gfCNCPoint3[26390] = {X 477.0833, Y 62.5348, Z -4.6667, A 0.000, B 0.000, C 0.000 }
gfCNCPoint3[26391] = {X 476.2899, Y 62.8890, Z -4.6667, A 0.000, B 0.000, C 0.000 }
gfCNCPoint3[26392] = {X 475.4402, Y 63.0707, Z -4.6667, A 0.000, B 0.000, C 0.000 }
gfCNCPoint3[26393] = {X 475.4407, Y 92.8975, Z -4.6667, A 0.000, B 0.000, C 0.000 }
gfCNCPoint3[26394] = {X 475.8927, Y 93.0046, Z -4.6667, A 0.000, B 0.000, C 0.000 }
gfCNCPoint3[26395] = {X 476.3374, Y 93.1385, Z -4.6667, A 0.000, B 0.000, C 0.000 }
gfCNCPoint3[26396] = {X 477.1187, Y 93.4937, Z -4.6667, A 0.000, B 0.000, C 0.000 }
gfCNCPoint3[26397] = {X 477.8098, Y 94.0025, Z -4.6667, A 0.000, B 0.000, C 0.000 }
gfCNCPoint3[26398] = {X 478.3809, Y 94.6431, Z -4.6667, A 0.000, B 0.000, C 0.000 }
gfCNCPoint3[26399] = {X 478.8074, Y 95.3878, Z -4.6667, A 0.000, B 0.000, C 0.000 }
gfCNCPoint3[26400] = {X 479.0709, Y 96.2046, Z -4.6667, A 0.000, B 0.000, C 0.000 }
gfCNCPoint3[26401] = {X 479.1600, Y 97.0582, Z -4.6667, A 0.000, B 0.000, C 0.000 }
gfCNCPoint3[26402] = {X 479.1600, Y 98.0000, Z -4.6667, A 0.000, B 0.000, C 0.000 }
gfCNCPoint3[26403] = {X 479.0557, Y 98.9257, Z -4.6667, A 0.000, B 0.000, C 0.000 }
gfCNCPoint3[26404] = {X 478.7480, Y 99.8050, Z -4.6667, A 0.000, B 0.000, C 0.000 }
gfCNCPoint3[26405] = {X 478.2524, Y 100.5937, Z -4.6667, A 0.000, B 0.000, C 0.000 }
gfCNCPoint3[26406] = {X 477.5937, Y 101.2524, Z -4.6667, A 0.000, B 0.000, C 0.000 }
gfCNCPoint3[26407] = {X 476.8050, Y 101.7480, Z -4.6667, A 0.000, B 0.000, C 0.000 }
gfCNCPoint3[26408] = {X 475.9257, Y 102.0557, Z -4.6667, A 0.000, B 0.000, C 0.000 }
gfCNCPoint3[26409] = {X 475.0000, Y 102.1600, Z -4.6667, A 0.000, B 0.000, C 0.000 }
gfCNCPoint3[26410] = {X 458.4596, Y 102.1600, Z -4.6667, A 0.000, B 0.000, C 0.000 }
gfCNCPoint3[26411] = {X 457.5339, Y 102.0557, Z -4.6667, A 0.000, B 0.000, C 0.000 }
gfCNCPoint3[26412] = {X 456.6546, Y 101.7480, Z -4.6667, A 0.000, B 0.000, C 0.000 }
gfCNCPoint3[26413] = {X 455.8659, Y 101.2524, Z -4.6667, A 0.000, B 0.000, C 0.000 }
gfCNCPoint3[26414] = {X 455.2072, Y 100.5937, Z -4.6667, A 0.000, B 0.000, C 0.000 }
gfCNCPoint3[26415] = {X 454.7116, Y 99.8050, Z -4.6667, A 0.000, B 0.000, C 0.000 }
gfCNCPoint3[26416] = {X 454.4039, Y 98.9257, Z -4.6667, A 0.000, B 0.000, C 0.000 }
gfCNCPoint3[26417] = {X 454.2996, Y 98.0000, Z -4.6667, A 0.000, B 0.000, C 0.000 }
gfCNCPoint3[26418] = {X 454.2996, Y 97.0659, Z -4.6667, A 0.000, B 0.000, C 0.000 }
gfCNCPoint3[26419] = {X 454.3903, Y 96.2022, Z -4.6667, A 0.000, B 0.000, C 0.000 }
gfCNCPoint3[26420] = {X 454.6583, Y 95.3761, Z -4.6667, A 0.000, B 0.000, C 0.000 }
gfCNCPoint3[26421] = {X 455.0920, Y 94.6237, Z -4.6667, A 0.000, B 0.000, C 0.000 }
gfCNCPoint3[26422] = {X 455.6724, Y 93.9777, Z -4.6667, A 0.000, B 0.000, C 0.000 }
gfCNCPoint3[26423] = {X 456.3743, Y 93.4663, Z -4.6667, A 0.000, B 0.000, C 0.000 }
gfCNCPoint3[26424] = {X 457.1672, Y 93.1118, Z -4.6667, A 0.000, B 0.000, C 0.000 }
gfCNCPoint3[26425] = {X 458.0163, Y 92.9296, Z -4.6667, A 0.000, B 0.000, C 0.000 }
gfCNCPoint3[26426] = {X 458.0163, Y 85.4858, Z -4.6667, A 0.000, B 0.000, C 0.000 }
gfCNCPoint3[26427] = {X 444.8411, Y 80.3211, Z -4.6667, A 0.000, B 0.000, C 0.000 }
gfCNCPoint3[26428] = {X 419.8629, Y 96.5017, Z -4.6667, A 0.000, B 0.000, C 0.000 }
gfCNCPoint3[26429] = {X 419.8667, Y 97.0654, Z -4.6667, A 0.000, B 0.000, C 0.000 }
gfCNCPoint3[26430] = {X 419.8667, Y 98.0000, Z -4.6667, A 0.000, B 0.000, C 0.000 }
gfCNCPoint3[26431] = {X 419.7624, Y 98.9257, Z -4.6667, A 0.000, B 0.000, C 0.000 }
gfCNCPoint3[26432] = {X 419.4547, Y 99.8050, Z -4.6667, A 0.000, B 0.000, C 0.000 }
gfCNCPoint3[26433] = {X 418.9591, Y 100.5937, Z -4.6667, A 0.000, B 0.000, C 0.000 }
gfCNCPoint3[26434] = {X 418.3004, Y 101.2524, Z -4.6667, A 0.000, B 0.000, C 0.000 }
gfCNCPoint3[26435] = {X 417.5117, Y 101.7480, Z -4.6667, A 0.000, B 0.000, C 0.000 }
gfCNCPoint3[26436] = {X 416.6324, Y 102.0557, Z -4.6667, A 0.000, B 0.000, C 0.000 }
gfCNCPoint3[26437] = {X 415.7067, Y 102.1600, Z -4.6667, A 0.000, B 0.000, C 0.000 }
gfCNCPoint3[26438] = {X 396.4059, Y 102.1600, Z -4.6667, A 0.000, B 0.000, C 0.000 }
gfCNCPoint3[26439] = {X 395.4803, Y 102.0557, Z -4.6667, A 0.000, B 0.000, C 0.000 }
gfCNCPoint3[26440] = {X 394.6010, Y 101.7480, Z -4.6667, A 0.000, B 0.000, C 0.000 }
gfCNCPoint3[26441] = {X 393.8122, Y 101.2524, Z -4.6667, A 0.000, B 0.000, C 0.000 }
gfCNCPoint3[26442] = {X 393.1535, Y 100.5937, Z -4.6667, A 0.000, B 0.000, C 0.000 }
gfCNCPoint3[26443] = {X 392.6579, Y 99.8050, Z -4.6667, A 0.000, B 0.000, C 0.000 }
gfCNCPoint3[26444] = {X 392.3502, Y 98.9257, Z -4.6667, A 0.000, B 0.000, C 0.000 }
gfCNCPoint3[26445] = {X 392.2459, Y 98.0000, Z -4.6667, A 0.000, B 0.000, C 0.000 }
gfCNCPoint3[26446] = {X 392.2459, Y 97.0659, Z -4.6667, A 0.000, B 0.000, C 0.000 }
gfCNCPoint3[26447] = {X 392.3511, Y 96.1365, Z -4.6667, A 0.000, B 0.000, C 0.000 }
gfCNCPoint3[26448] = {X 392.6612, Y 95.2541, Z -4.6667, A 0.000, B 0.000, C 0.000 }
gfCNCPoint3[26449] = {X 393.1607, Y 94.4633, Z -4.6667, A 0.000, B 0.000, C 0.000 }
gfCNCPoint3[26450] = {X 393.8242, Y 93.8040, Z -4.6667, A 0.000, B 0.000, C 0.000 }
gfCNCPoint3[26451] = {X 394.6182, Y 93.3096, Z -4.6667, A 0.000, B 0.000, C 0.000 }
gfCNCPoint3[26452] = {X 395.5026, Y 93.0052, Z -4.6667, A 0.000, B 0.000, C 0.000 }
gfCNCPoint3[26453] = {X 396.4327, Y 92.9060, Z -4.6667, A 0.000, B 0.000, C 0.000 }
gfCNCPoint3[26454] = {X 397.3745, Y 92.8625, Z -4.6667, A 0.000, B 0.000, C 0.000 }
gfCNCPoint3[26455] = {X 398.3131, Y 92.7731, Z -4.6667, A 0.000, B 0.000, C 0.000 }
gfCNCPoint3[26456] = {X 398.9990, Y 92.6067, Z -4.6667, A 0.000, B 0.000, C 0.000 }
gfCNCPoint3[26457] = {X 399.6307, Y 92.2919, Z -4.6667, A 0.000, B 0.000, C 0.000 }
gfCNCPoint3[26458] = {X 413.8854, Y 83.1633, Z -4.6667, A 0.000, B 0.000, C 0.000 }
gfCNCPoint3[26459] = {X 411.7283, Y 79.7948, Z -4.6667, A 0.000, B 0.000, C 0.000 }
gfCNCPoint3[26460] = {X 413.9286, Y 83.2307, Z -4.6667, A 0.000, B 0.000, C 0.000 }
gfCNCPoint3[26461] = {X 428.5801, Y 73.8479, Z -4.6667, A 0.000, B 0.000, C 0.000 }
gfCNCPoint3[26462] = {X 403.8433, Y 64.1425, Z -4.6667, A 0.000, B 0.000, C 0.000 }
gfCNCPoint3[26463] = {X 402.1208, Y 63.5723, Z -4.6667, A 0.000, B 0.000, C 0.000 }
gfCNCPoint3[26464] = {X 400.3462, Y 63.1946, Z -4.6667, A 0.000, B 0.000, C 0.000 }
gfCNCPoint3[26465] = {X 398.5408, Y 63.0140, Z -4.6667, A 0.000, B 0.000, C 0.000 }
gfCNCPoint3[26466] = {X 397.6404, Y 62.9096, Z -4.6667, A 0.000, B 0.000, C 0.000 }
gfCNCPoint3[26467] = {X 396.7852, Y 62.6089, Z -4.6667, A 0.000, B 0.000, C 0.000 }
gfCNCPoint3[26468] = {X 396.0176, Y 62.1269, Z -4.6667, A 0.000, B 0.000, C 0.000 }
gfCNCPoint3[26469] = {X 395.3753, Y 61.4873, Z -4.6667, A 0.000, B 0.000, C 0.000 }
gfCNCPoint3[26470] = {X 394.8902, Y 60.7216, Z -4.6667, A 0.000, B 0.000, C 0.000 }
gfCNCPoint3[26471] = {X 394.5860, Y 59.8677, Z -4.6667, A 0.000, B 0.000, C 0.000 }
gfCNCPoint3[26472] = {X 394.4779, Y 58.9678, Z -4.6667, A 0.000, B 0.000, C 0.000 }
gfCNCPoint3[26473] = {X 394.4777, Y 58.0000, Z -4.6667, A 0.000, B 0.000, C 0.000 }
gfCNCPoint3[26474] = {X 394.5800, Y 57.0921, Z -4.6667, A 0.000, B 0.000, C 0.000 }
gfCNCPoint3[26475] = {X 394.8818, Y 56.2298, Z -4.6667, A 0.000, B 0.000, C 0.000 }
gfCNCPoint3[26476] = {X 395.3678, Y 55.4562, Z -4.6667, A 0.000, B 0.000, C 0.000 }
gfCNCPoint3[26477] = {X 396.0139, Y 54.8101, Z -4.6667, A 0.000, B 0.000, C 0.000 }
gfCNCPoint3[26478] = {X 396.7875, Y 54.3240, Z -4.6667, A 0.000, B 0.000, C 0.000 }
gfCNCPoint3[26479] = {X 397.6498, Y 54.0223, Z -4.6667, A 0.000, B 0.000, C 0.000 }
gfCNCPoint3[26480] = {X 398.5577, Y 53.9200, Z -4.6667, A 0.000, B 0.000, C 0.000 }
gfCNCPoint3[26481] = {X 419.4886, Y 53.9200, Z -4.6667, A 0.000, B 0.000, C 0.000 }
gfCNCPoint3[26482] = {X 420.3965, Y 54.0223, Z -4.6667, A 0.000, B 0.000, C 0.000 }
gfCNCPoint3[26483] = {X 421.2588, Y 54.3240, Z -4.6667, A 0.000, B 0.000, C 0.000 }
gfCNCPoint3[26484] = {X 422.0324, Y 54.8101, Z -4.6667, A 0.000, B 0.000, C 0.000 }
gfCNCPoint3[26485] = {X 422.6785, Y 55.4562, Z -4.6667, A 0.000, B 0.000, C 0.000 }
gfCNCPoint3[26486] = {X 423.1646, Y 56.2298, Z -4.6667, A 0.000, B 0.000, C 0.000 }
gfCNCPoint3[26487] = {X 423.4663, Y 57.0921, Z -4.6667, A 0.000, B 0.000, C 0.000 }
gfCNCPoint3[26488] = {X 423.5686, Y 58.0000, Z -4.6667, A 0.000, B 0.000, C 0.000 }
gfCNCPoint3[26489] = {X 423.5686, Y 58.3962, Z -4.6667, A 0.000, B 0.000, C 0.000 }
gfCNCPoint3[26490] = {X 429.5238, Y 60.7167, Z -4.6667, A 0.000, B 0.000, C 0.000 }
gfCNCPoint3[26491] = {X 458.0985, Y 72.0540, Z -4.6667, A 0.000, B 0.000, C 0.000 }
gfCNCPoint3[26492] = {X 458.1008, Y 62.9983, Z -4.6667, A 0.000, B 0.000, C 0.000 }
gfCNCPoint3[26493] = {X 457.9644, Y 62.9839, Z -4.6667, A 0.000, B 0.000, C 0.000 }
gfCNCPoint3[26494] = {X 457.8285, Y 62.9650, Z -4.6667, A 0.000, B 0.000, C 0.000 }
gfCNCPoint3[26495] = {X 456.9091, Y 62.7079, Z -4.6667, A 0.000, B 0.000, C 0.000 }
gfCNCPoint3[26496] = {X 456.0745, Y 62.2443, Z -4.6667, A 0.000, B 0.000, C 0.000 }
gfCNCPoint3[26497] = {X 455.3705, Y 61.5994, Z -4.6667, A 0.000, B 0.000, C 0.000 }
gfCNCPoint3[26498] = {X 454.8357, Y 60.8085, Z -4.6667, A 0.000, B 0.000, C 0.000 }
gfCNCPoint3[26499] = {X 454.4993, Y 59.9150, Z -4.6667, A 0.000, B 0.000, C 0.000 }
gfCNCPoint3[26500] = {X 454.3797, Y 58.9678, Z -4.6667, A 0.000, B 0.000, C 0.000 }
gfCNCPoint3[26501] = {X 454.3796, Y 58.0000, Z -4.6667, A 0.000, B 0.000, C 0.000 }
gfCNCPoint3[26502] = {X 454.4819, Y 57.0921, Z -4.6667, A 0.000, B 0.000, C 0.000 }
gfCNCPoint3[26503] = {X 454.7837, Y 56.2298, Z -4.6667, A 0.000, B 0.000, C 0.000 }
gfCNCPoint3[26504] = {X 455.2697, Y 55.4562, Z -4.6667, A 0.000, B 0.000, C 0.000 }
gfCNCPoint3[26505] = {X 455.9158, Y 54.8101, Z -4.6667, A 0.000, B 0.000, C 0.000 }
gfCNCPoint3[26506] = {X 456.6894, Y 54.3240, Z -4.6667, A 0.000, B 0.000, C 0.000 }
gfCNCPoint3[26507] = {X 457.5517, Y 54.0223, Z -4.6667, A 0.000, B 0.000, C 0.000 }
gfCNCPoint3[26508] = {X 458.4596, Y 53.9200, Z -4.6667, A 0.000, B 0.000, C 0.000 }
gfCNCPoint3[26509] = {X 475.0000, Y 53.9200, Z -4.6667, A 0.000, B 0.000, C 0.000 }
gfCNCPoint3[26510] = {X 475.9079, Y 54.0223, Z -4.6667, A 0.000, B 0.000, C 0.000 }
gfCNCPoint3[26511] = {X 476.7702, Y 54.3240, Z -4.6667, A 0.000, B 0.000, C 0.000 }
gfCNCPoint3[26512] = {X 477.5438, Y 54.8101, Z -4.6667, A 0.000, B 0.000, C 0.000 }
gfCNCPoint3[26513] = {X 478.1899, Y 55.4562, Z -4.6667, A 0.000, B 0.000, C 0.000 }
gfCNCPoint3[26514] = {X 478.6760, Y 56.2298, Z -4.6667, A 0.000, B 0.000, C 0.000 }
gfCNCPoint3[26515] = {X 478.9777, Y 57.0921, Z -4.6667, A 0.000, B 0.000, C 0.000 }
gfCNCPoint3[26516] = {X 479.0800, Y 58.0000, Z -4.6667, A 0.000, B 0.000, C 0.000 }
gfCNCPoint3[26517] = {X 479.0800, Y 58.9342, Z -4.6667, A 0.000, B 0.000, C 0.000 }
gfCNCPoint3[26518] = {X 478.9888, Y 59.7918, Z -4.6667, A 0.000, B 0.000, C 0.000 }
gfCNCPoint3[26519] = {X 478.7194, Y 60.6110, Z -4.6667, A 0.000, B 0.000, C 0.000 }
gfCNCPoint3[26520] = {X 478.2839, Y 61.3553, Z -4.6667, A 0.000, B 0.000, C 0.000 }
gfCNCPoint3[26521] = {X 477.7016, Y 61.9915, Z -4.6667, A 0.000, B 0.000, C 0.000 }
gfCNCPoint3[26522] = {X 476.9986, Y 62.4910, Z -4.6667, A 0.000, B 0.000, C 0.000 }
gfCNCPoint3[26523] = {X 476.2064, Y 62.8316, Z -4.6667, A 0.000, B 0.000, C 0.000 }
gfCNCPoint3[26524] = {X 475.3602, Y 62.9981, Z -4.6667, A 0.000, B 0.000, C 0.000 }
gfCNCPoint3[26525] = {X 475.3607, Y 92.9630, Z -4.6667, A 0.000, B 0.000, C 0.000 }
gfCNCPoint3[26526] = {X 475.8404, Y 93.0734, Z -4.6667, A 0.000, B 0.000, C 0.000 }
gfCNCPoint3[26527] = {X 476.3121, Y 93.2144, Z -4.6667, A 0.000, B 0.000, C 0.000 }
gfCNCPoint3[26528] = {X 477.0782, Y 93.5627, Z -4.6667, A 0.000, B 0.000, C 0.000 }
gfCNCPoint3[26529] = {X 477.7560, Y 94.0616, Z -4.6667, A 0.000, B 0.000, C 0.000 }
gfCNCPoint3[26530] = {X 478.3160, Y 94.6898, Z -4.6667, A 0.000, B 0.000, C 0.000 }
gfCNCPoint3[26531] = {X 478.7342, Y 95.4202, Z -4.6667, A 0.000, B 0.000, C 0.000 }
gfCNCPoint3[26532] = {X 478.9926, Y 96.2211, Z -4.6667, A 0.000, B 0.000, C 0.000 }
gfCNCPoint3[26533] = {X 479.0800, Y 97.0582, Z -4.6667, A 0.000, B 0.000, C 0.000 }
gfCNCPoint3[26534] = {X 479.0800, Y 98.0000, Z -4.6667, A 0.000, B 0.000, C 0.000 }
gfCNCPoint3[26535] = {X 478.9777, Y 98.9079, Z -4.6667, A 0.000, B 0.000, C 0.000 }
gfCNCPoint3[26536] = {X 478.6760, Y 99.7702, Z -4.6667, A 0.000, B 0.000, C 0.000 }
gfCNCPoint3[26537] = {X 478.1899, Y 100.5438, Z -4.6667, A 0.000, B 0.000, C 0.000 }
gfCNCPoint3[26538] = {X 477.5438, Y 101.1899, Z -4.6667, A 0.000, B 0.000, C 0.000 }
gfCNCPoint3[26539] = {X 476.7702, Y 101.6760, Z -4.6667, A 0.000, B 0.000, C 0.000 }
gfCNCPoint3[26540] = {X 475.9079, Y 101.9777, Z -4.6667, A 0.000, B 0.000, C 0.000 }
gfCNCPoint3[26541] = {X 475.0000, Y 102.0800, Z -4.6667, A 0.000, B 0.000, C 0.000 }
gfCNCPoint3[26542] = {X 458.4596, Y 102.0800, Z -4.6667, A 0.000, B 0.000, C 0.000 }
gfCNCPoint3[26543] = {X 457.5517, Y 101.9777, Z -4.6667, A 0.000, B 0.000, C 0.000 }
gfCNCPoint3[26544] = {X 456.6894, Y 101.6760, Z -4.6667, A 0.000, B 0.000, C 0.000 }
gfCNCPoint3[26545] = {X 455.9158, Y 101.1899, Z -4.6667, A 0.000, B 0.000, C 0.000 }
gfCNCPoint3[26546] = {X 455.2697, Y 100.5438, Z -4.6667, A 0.000, B 0.000, C 0.000 }
gfCNCPoint3[26547] = {X 454.7837, Y 99.7702, Z -4.6667, A 0.000, B 0.000, C 0.000 }
gfCNCPoint3[26548] = {X 454.4819, Y 98.9079, Z -4.6667, A 0.000, B 0.000, C 0.000 }
gfCNCPoint3[26549] = {X 454.3796, Y 98.0000, Z -4.6667, A 0.000, B 0.000, C 0.000 }
gfCNCPoint3[26550] = {X 454.3796, Y 97.0659, Z -4.6667, A 0.000, B 0.000, C 0.000 }
gfCNCPoint3[26551] = {X 454.4707, Y 96.2088, Z -4.6667, A 0.000, B 0.000, C 0.000 }
gfCNCPoint3[26552] = {X 454.7398, Y 95.3899, Z -4.6667, A 0.000, B 0.000, C 0.000 }
gfCNCPoint3[26553] = {X 455.1749, Y 94.6458, Z -4.6667, A 0.000, B 0.000, C 0.000 }
gfCNCPoint3[26554] = {X 455.7566, Y 94.0098, Z -4.6667, A 0.000, B 0.000, C 0.000 }
gfCNCPoint3[26555] = {X 456.4590, Y 93.5101, Z -4.6667, A 0.000, B 0.000, C 0.000 }
gfCNCPoint3[26556] = {X 457.2507, Y 93.1692, Z -4.6667, A 0.000, B 0.000, C 0.000 }
gfCNCPoint3[26557] = {X 458.0963, Y 93.0021, Z -4.6667, A 0.000, B 0.000, C 0.000 }
gfCNCPoint3[26558] = {X 458.0963, Y 85.4313, Z -4.6667, A 0.000, B 0.000, C 0.000 }
gfCNCPoint3[26559] = {X 444.8320, Y 80.2317, Z -4.6667, A 0.000, B 0.000, C 0.000 }
gfCNCPoint3[26560] = {X 419.7826, Y 96.4583, Z -4.6667, A 0.000, B 0.000, C 0.000 }
gfCNCPoint3[26561] = {X 419.7867, Y 97.0656, Z -4.6667, A 0.000, B 0.000, C 0.000 }
gfCNCPoint3[26562] = {X 419.7867, Y 98.0000, Z -4.6667, A 0.000, B 0.000, C 0.000 }
gfCNCPoint3[26563] = {X 419.6844, Y 98.9079, Z -4.6667, A 0.000, B 0.000, C 0.000 }
gfCNCPoint3[26564] = {X 419.3827, Y 99.7702, Z -4.6667, A 0.000, B 0.000, C 0.000 }
gfCNCPoint3[26565] = {X 418.8966, Y 100.5438, Z -4.6667, A 0.000, B 0.000, C 0.000 }
gfCNCPoint3[26566] = {X 418.2505, Y 101.1899, Z -4.6667, A 0.000, B 0.000, C 0.000 }
gfCNCPoint3[26567] = {X 417.4769, Y 101.6760, Z -4.6667, A 0.000, B 0.000, C 0.000 }
gfCNCPoint3[26568] = {X 416.6146, Y 101.9777, Z -4.6667, A 0.000, B 0.000, C 0.000 }
gfCNCPoint3[26569] = {X 415.7067, Y 102.0800, Z -4.6667, A 0.000, B 0.000, C 0.000 }
gfCNCPoint3[26570] = {X 396.4059, Y 102.0800, Z -4.6667, A 0.000, B 0.000, C 0.000 }
gfCNCPoint3[26571] = {X 395.4981, Y 101.9777, Z -4.6667, A 0.000, B 0.000, C 0.000 }
gfCNCPoint3[26572] = {X 394.6357, Y 101.6760, Z -4.6667, A 0.000, B 0.000, C 0.000 }
gfCNCPoint3[26573] = {X 393.8621, Y 101.1899, Z -4.6667, A 0.000, B 0.000, C 0.000 }
gfCNCPoint3[26574] = {X 393.2161, Y 100.5438, Z -4.6667, A 0.000, B 0.000, C 0.000 }
gfCNCPoint3[26575] = {X 392.7300, Y 99.7702, Z -4.6667, A 0.000, B 0.000, C 0.000 }
gfCNCPoint3[26576] = {X 392.4282, Y 98.9079, Z -4.6667, A 0.000, B 0.000, C 0.000 }
gfCNCPoint3[26577] = {X 392.3259, Y 98.0000, Z -4.6667, A 0.000, B 0.000, C 0.000 }
gfCNCPoint3[26578] = {X 392.3259, Y 97.0659, Z -4.6667, A 0.000, B 0.000, C 0.000 }
gfCNCPoint3[26579] = {X 392.4291, Y 96.1542, Z -4.6667, A 0.000, B 0.000, C 0.000 }
gfCNCPoint3[26580] = {X 392.7334, Y 95.2886, Z -4.6667, A 0.000, B 0.000, C 0.000 }
gfCNCPoint3[26581] = {X 393.2234, Y 94.5129, Z -4.6667, A 0.000, B 0.000, C 0.000 }
gfCNCPoint3[26582] = {X 393.8744, Y 93.8663, Z -4.6667, A 0.000, B 0.000, C 0.000 }
gfCNCPoint3[26583] = {X 394.6533, Y 93.3815, Z -4.6667, A 0.000, B 0.000, C 0.000 }
gfCNCPoint3[26584] = {X 395.5210, Y 93.0831, Z -4.6667, A 0.000, B 0.000, C 0.000 }
gfCNCPoint3[26585] = {X 396.4333, Y 92.9860, Z -4.6667, A 0.000, B 0.000, C 0.000 }
gfCNCPoint3[26586] = {X 397.3798, Y 92.9423, Z -4.6667, A 0.000, B 0.000, C 0.000 }
gfCNCPoint3[26587] = {X 398.3229, Y 92.8525, Z -4.6667, A 0.000, B 0.000, C 0.000 }
gfCNCPoint3[26588] = {X 399.0264, Y 92.6819, Z -4.6667, A 0.000, B 0.000, C 0.000 }
gfCNCPoint3[26589] = {X 399.6742, Y 92.3590, Z -4.6667, A 0.000, B 0.000, C 0.000 }
gfCNCPoint3[26590] = {X 413.9286, Y 83.2307, Z -4.6667, A 0.000, B 0.000, C 0.000 }
gfCNCPoint3[26591] = {X 411.7650, Y 79.8521, Z -4.6667, A 0.000, B 0.000, C 0.000 }
gfCNCPoint3[26592] = {X 411.7673, Y 79.8506, Z -4.6667, A 0.000, B 0.000, C 0.000 }
gfCNCPoint3[26593] = {X 413.9652, Y 83.2880, Z -4.6667, A 0.000, B 0.000, C 0.000 }
gfCNCPoint3[26594] = {X 428.7554, Y 73.8308, Z -4.6667, A 0.000, B 0.000, C 0.000 }
gfCNCPoint3[26595] = {X 403.8726, Y 64.0680, Z -4.6667, A 0.000, B 0.000, C 0.000 }
gfCNCPoint3[26596] = {X 402.1412, Y 63.4949, Z -4.6667, A 0.000, B 0.000, C 0.000 }
gfCNCPoint3[26597] = {X 400.3574, Y 63.1154, Z -4.6667, A 0.000, B 0.000, C 0.000 }
gfCNCPoint3[26598] = {X 398.5427, Y 62.9340, Z -4.6667, A 0.000, B 0.000, C 0.000 }
gfCNCPoint3[26599] = {X 397.6551, Y 62.8309, Z -4.6667, A 0.000, B 0.000, C 0.000 }
gfCNCPoint3[26600] = {X 396.8125, Y 62.5333, Z -4.6667, A 0.000, B 0.000, C 0.000 }
gfCNCPoint3[26601] = {X 396.0571, Y 62.0560, Z -4.6667, A 0.000, B 0.000, C 0.000 }
gfCNCPoint3[26602] = {X 395.4264, Y 61.4230, Z -4.6667, A 0.000, B 0.000, C 0.000 }
gfCNCPoint3[26603] = {X 394.9520, Y 60.6657, Z -4.6667, A 0.000, B 0.000, C 0.000 }
gfCNCPoint3[26604] = {X 394.6575, Y 59.8220, Z -4.6667, A 0.000, B 0.000, C 0.000 }
gfCNCPoint3[26605] = {X 394.5577, Y 58.9341, Z -4.6667, A 0.000, B 0.000, C 0.000 }
gfCNCPoint3[26606] = {X 394.5577, Y 58.0000, Z -4.6667, A 0.000, B 0.000, C 0.000 }
gfCNCPoint3[26607] = {X 394.6580, Y 57.1099, Z -4.6667, A 0.000, B 0.000, C 0.000 }
gfCNCPoint3[26608] = {X 394.9538, Y 56.2645, Z -4.6667, A 0.000, B 0.000, C 0.000 }
gfCNCPoint3[26609] = {X 395.4304, Y 55.5060, Z -4.6667, A 0.000, B 0.000, C 0.000 }
gfCNCPoint3[26610] = {X 396.0638, Y 54.8727, Z -4.6667, A 0.000, B 0.000, C 0.000 }
gfCNCPoint3[26611] = {X 396.8222, Y 54.3961, Z -4.6667, A 0.000, B 0.000, C 0.000 }
gfCNCPoint3[26612] = {X 397.6676, Y 54.1003, Z -4.6667, A 0.000, B 0.000, C 0.000 }
gfCNCPoint3[26613] = {X 398.5577, Y 54.0000, Z -4.6667, A 0.000, B 0.000, C 0.000 }
gfCNCPoint3[26614] = {X 419.4886, Y 54.0000, Z -4.6667, A 0.000, B 0.000, C 0.000 }
gfCNCPoint3[26615] = {X 420.3787, Y 54.1003, Z -4.6667, A 0.000, B 0.000, C 0.000 }
gfCNCPoint3[26616] = {X 421.2241, Y 54.3961, Z -4.6667, A 0.000, B 0.000, C 0.000 }
gfCNCPoint3[26617] = {X 421.9826, Y 54.8727, Z -4.6667, A 0.000, B 0.000, C 0.000 }
gfCNCPoint3[26618] = {X 422.6159, Y 55.5060, Z -4.6667, A 0.000, B 0.000, C 0.000 }
gfCNCPoint3[26619] = {X 423.0925, Y 56.2645, Z -4.6667, A 0.000, B 0.000, C 0.000 }
gfCNCPoint3[26620] = {X 423.3883, Y 57.1099, Z -4.6667, A 0.000, B 0.000, C 0.000 }
gfCNCPoint3[26621] = {X 423.4886, Y 58.0000, Z -4.6667, A 0.000, B 0.000, C 0.000 }
gfCNCPoint3[26622] = {X 423.4886, Y 58.4509, Z -4.6667, A 0.000, B 0.000, C 0.000 }
gfCNCPoint3[26623] = {X 429.4945, Y 60.7912, Z -4.6667, A 0.000, B 0.000, C 0.000 }
gfCNCPoint3[26624] = {X 458.1785, Y 72.1718, Z -4.6667, A 0.000, B 0.000, C 0.000 }
gfCNCPoint3[26625] = {X 458.1791, Y 63.0387, Z -4.6667, A 0.000, B 0.000, C 0.000 }
gfCNCPoint3[26626] = {X 458.1841, Y 62.9246, Z -4.6667, A 0.000, B 0.000, C 0.000 }
gfCNCPoint3[26627] = {X 458.0121, Y 62.9090, Z -4.6667, A 0.000, B 0.000, C 0.000 }
gfCNCPoint3[26628] = {X 457.8409, Y 62.8859, Z -4.6667, A 0.000, B 0.000, C 0.000 }
gfCNCPoint3[26629] = {X 456.9344, Y 62.6319, Z -4.6667, A 0.000, B 0.000, C 0.000 }
gfCNCPoint3[26630] = {X 456.1123, Y 62.1729, Z -4.6667, A 0.000, B 0.000, C 0.000 }
gfCNCPoint3[26631] = {X 455.4203, Y 61.5346, Z -4.6667, A 0.000, B 0.000, C 0.000 }
gfCNCPoint3[26632] = {X 454.8967, Y 60.7521, Z -4.6667, A 0.000, B 0.000, C 0.000 }
gfCNCPoint3[26633] = {X 454.5704, Y 59.8690, Z -4.6667, A 0.000, B 0.000, C 0.000 }
gfCNCPoint3[26634] = {X 454.4596, Y 58.9341, Z -4.6667, A 0.000, B 0.000, C 0.000 }
gfCNCPoint3[26635] = {X 454.4596, Y 58.0000, Z -4.6667, A 0.000, B 0.000, C 0.000 }
gfCNCPoint3[26636] = {X 454.5599, Y 57.1099, Z -4.6667, A 0.000, B 0.000, C 0.000 }
gfCNCPoint3[26637] = {X 454.8557, Y 56.2645, Z -4.6667, A 0.000, B 0.000, C 0.000 }
gfCNCPoint3[26638] = {X 455.3323, Y 55.5060, Z -4.6667, A 0.000, B 0.000, C 0.000 }
gfCNCPoint3[26639] = {X 455.9656, Y 54.8727, Z -4.6667, A 0.000, B 0.000, C 0.000 }
gfCNCPoint3[26640] = {X 456.7241, Y 54.3961, Z -4.6667, A 0.000, B 0.000, C 0.000 }
gfCNCPoint3[26641] = {X 457.5695, Y 54.1003, Z -4.6667, A 0.000, B 0.000, C 0.000 }
gfCNCPoint3[26642] = {X 458.4596, Y 54.0000, Z -4.6667, A 0.000, B 0.000, C 0.000 }
gfCNCPoint3[26643] = {X 475.0000, Y 54.0000, Z -4.6667, A 0.000, B 0.000, C 0.000 }
gfCNCPoint3[26644] = {X 475.8901, Y 54.1003, Z -4.6667, A 0.000, B 0.000, C 0.000 }
gfCNCPoint3[26645] = {X 476.7355, Y 54.3961, Z -4.6667, A 0.000, B 0.000, C 0.000 }
gfCNCPoint3[26646] = {X 477.4940, Y 54.8727, Z -4.6667, A 0.000, B 0.000, C 0.000 }
gfCNCPoint3[26647] = {X 478.1273, Y 55.5060, Z -4.6667, A 0.000, B 0.000, C 0.000 }
gfCNCPoint3[26648] = {X 478.6039, Y 56.2645, Z -4.6667, A 0.000, B 0.000, C 0.000 }
gfCNCPoint3[26649] = {X 478.8997, Y 57.1099, Z -4.6667, A 0.000, B 0.000, C 0.000 }
gfCNCPoint3[26650] = {X 479.0000, Y 58.0000, Z -4.6667, A 0.000, B 0.000, C 0.000 }
gfCNCPoint3[26651] = {X 478.9999, Y 58.9671, Z -4.6667, A 0.000, B 0.000, C 0.000 }
gfCNCPoint3[26652] = {X 478.9023, Y 59.8127, Z -4.6667, A 0.000, B 0.000, C 0.000 }
gfCNCPoint3[26653] = {X 478.6280, Y 60.6185, Z -4.6667, A 0.000, B 0.000, C 0.000 }
gfCNCPoint3[26654] = {X 478.1895, Y 61.3480, Z -4.6667, A 0.000, B 0.000, C 0.000 }
gfCNCPoint3[26655] = {X 477.6065, Y 61.9682, Z -4.6667, A 0.000, B 0.000, C 0.000 }
gfCNCPoint3[26656] = {X 476.9055, Y 62.4510, Z -4.6667, A 0.000, B 0.000, C 0.000 }
gfCNCPoint3[26657] = {X 476.1182, Y 62.7746, Z -4.6667, A 0.000, B 0.000, C 0.000 }
gfCNCPoint3[26658] = {X 475.2802, Y 62.9242, Z -4.6667, A 0.000, B 0.000, C 0.000 }
gfCNCPoint3[26659] = {X 475.2807, Y 93.0291, Z -4.6667, A 0.000, B 0.000, C 0.000 }
gfCNCPoint3[26660] = {X 475.7882, Y 93.1424, Z -4.6667, A 0.000, B 0.000, C 0.000 }
gfCNCPoint3[26661] = {X 476.2867, Y 93.2903, Z -4.6667, A 0.000, B 0.000, C 0.000 }
gfCNCPoint3[26662] = {X 477.0377, Y 93.6317, Z -4.6667, A 0.000, B 0.000, C 0.000 }
gfCNCPoint3[26663] = {X 477.7021, Y 94.1208, Z -4.6667, A 0.000, B 0.000, C 0.000 }
gfCNCPoint3[26664] = {X 478.2511, Y 94.7366, Z -4.6667, A 0.000, B 0.000, C 0.000 }
gfCNCPoint3[26665] = {X 478.6611, Y 95.4525, Z -4.6667, A 0.000, B 0.000, C 0.000 }
gfCNCPoint3[26666] = {X 478.9143, Y 96.2377, Z -4.6667, A 0.000, B 0.000, C 0.000 }
gfCNCPoint3[26667] = {X 479.0000, Y 97.0582, Z -4.6667, A 0.000, B 0.000, C 0.000 }
gfCNCPoint3[26668] = {X 479.0000, Y 98.0000, Z -4.6667, A 0.000, B 0.000, C 0.000 }
gfCNCPoint3[26669] = {X 478.8997, Y 98.8901, Z -4.6667, A 0.000, B 0.000, C 0.000 }
gfCNCPoint3[26670] = {X 478.6039, Y 99.7355, Z -4.6667, A 0.000, B 0.000, C 0.000 }
gfCNCPoint3[26671] = {X 478.1273, Y 100.4940, Z -4.6667, A 0.000, B 0.000, C 0.000 }
gfCNCPoint3[26672] = {X 477.4940, Y 101.1273, Z -4.6667, A 0.000, B 0.000, C 0.000 }
gfCNCPoint3[26673] = {X 476.7355, Y 101.6039, Z -4.6667, A 0.000, B 0.000, C 0.000 }
gfCNCPoint3[26674] = {X 475.8901, Y 101.8997, Z -4.6667, A 0.000, B 0.000, C 0.000 }
gfCNCPoint3[26675] = {X 475.0000, Y 102.0000, Z -4.6667, A 0.000, B 0.000, C 0.000 }
gfCNCPoint3[26676] = {X 458.4596, Y 102.0000, Z -4.6667, A 0.000, B 0.000, C 0.000 }
gfCNCPoint3[26677] = {X 457.5695, Y 101.8997, Z -4.6667, A 0.000, B 0.000, C 0.000 }
gfCNCPoint3[26678] = {X 456.7241, Y 101.6039, Z -4.6667, A 0.000, B 0.000, C 0.000 }
gfCNCPoint3[26679] = {X 455.9656, Y 101.1273, Z -4.6667, A 0.000, B 0.000, C 0.000 }
gfCNCPoint3[26680] = {X 455.3323, Y 100.4940, Z -4.6667, A 0.000, B 0.000, C 0.000 }
gfCNCPoint3[26681] = {X 454.8557, Y 99.7355, Z -4.6667, A 0.000, B 0.000, C 0.000 }
gfCNCPoint3[26682] = {X 454.5599, Y 98.8901, Z -4.6667, A 0.000, B 0.000, C 0.000 }
gfCNCPoint3[26683] = {X 454.4596, Y 98.0000, Z -4.6667, A 0.000, B 0.000, C 0.000 }
gfCNCPoint3[26684] = {X 454.4596, Y 97.0659, Z -4.6667, A 0.000, B 0.000, C 0.000 }
gfCNCPoint3[26685] = {X 454.5511, Y 96.2154, Z -4.6667, A 0.000, B 0.000, C 0.000 }
gfCNCPoint3[26686] = {X 454.8213, Y 95.4037, Z -4.6667, A 0.000, B 0.000, C 0.000 }
gfCNCPoint3[26687] = {X 455.2580, Y 94.6681, Z -4.6667, A 0.000, B 0.000, C 0.000 }
gfCNCPoint3[26688] = {X 455.8411, Y 94.0422, Z -4.6667, A 0.000, B 0.000, C 0.000 }
gfCNCPoint3[26689] = {X 456.5439, Y 93.5545, Z -4.6667, A 0.000, B 0.000, C 0.000 }
gfCNCPoint3[26690] = {X 457.3344, Y 93.2275, Z -4.6667, A 0.000, B 0.000, C 0.000 }
gfCNCPoint3[26691] = {X 458.1763, Y 93.0760, Z -4.6667, A 0.000, B 0.000, C 0.000 }
gfCNCPoint3[26692] = {X 458.1763, Y 85.3767, Z -4.6667, A 0.000, B 0.000, C 0.000 }
gfCNCPoint3[26693] = {X 445.0142, Y 80.2171, Z -4.6667, A 0.000, B 0.000, C 0.000 }
gfCNCPoint3[26694] = {X 444.8241, Y 80.1415, Z -4.6667, A 0.000, B 0.000, C 0.000 }
gfCNCPoint3[26695] = {X 419.7023, Y 96.4150, Z -4.6667, A 0.000, B 0.000, C 0.000 }
gfCNCPoint3[26696] = {X 419.7067, Y 97.0659, Z -4.6667, A 0.000, B 0.000, C 0.000 }
gfCNCPoint3[26697] = {X 419.7067, Y 98.0000, Z -4.6667, A 0.000, B 0.000, C 0.000 }
gfCNCPoint3[26698] = {X 419.6064, Y 98.8901, Z -4.6667, A 0.000, B 0.000, C 0.000 }
gfCNCPoint3[26699] = {X 419.3106, Y 99.7355, Z -4.6667, A 0.000, B 0.000, C 0.000 }
gfCNCPoint3[26700] = {X 418.8340, Y 100.4940, Z -4.6667, A 0.000, B 0.000, C 0.000 }
gfCNCPoint3[26701] = {X 418.2007, Y 101.1273, Z -4.6667, A 0.000, B 0.000, C 0.000 }
gfCNCPoint3[26702] = {X 417.4422, Y 101.6039, Z -4.6667, A 0.000, B 0.000, C 0.000 }
gfCNCPoint3[26703] = {X 416.5968, Y 101.8997, Z -4.6667, A 0.000, B 0.000, C 0.000 }
gfCNCPoint3[26704] = {X 415.7067, Y 102.0000, Z -4.6667, A 0.000, B 0.000, C 0.000 }
gfCNCPoint3[26705] = {X 396.4059, Y 102.0000, Z -4.6667, A 0.000, B 0.000, C 0.000 }
gfCNCPoint3[26706] = {X 395.5159, Y 101.8997, Z -4.6667, A 0.000, B 0.000, C 0.000 }
gfCNCPoint3[26707] = {X 394.6704, Y 101.6039, Z -4.6667, A 0.000, B 0.000, C 0.000 }
gfCNCPoint3[26708] = {X 393.9120, Y 101.1273, Z -4.6667, A 0.000, B 0.000, C 0.000 }
gfCNCPoint3[26709] = {X 393.2786, Y 100.4940, Z -4.6667, A 0.000, B 0.000, C 0.000 }
gfCNCPoint3[26710] = {X 392.8021, Y 99.7355, Z -4.6667, A 0.000, B 0.000, C 0.000 }
gfCNCPoint3[26711] = {X 392.5062, Y 98.8901, Z -4.6667, A 0.000, B 0.000, C 0.000 }
gfCNCPoint3[26712] = {X 392.4059, Y 98.0000, Z -4.6667, A 0.000, B 0.000, C 0.000 }
gfCNCPoint3[26713] = {X 392.4059, Y 97.0659, Z -4.6667, A 0.000, B 0.000, C 0.000 }
gfCNCPoint3[26714] = {X 392.5071, Y 96.1720, Z -4.6667, A 0.000, B 0.000, C 0.000 }
gfCNCPoint3[26715] = {X 392.8056, Y 95.3232, Z -4.6667, A 0.000, B 0.000, C 0.000 }
gfCNCPoint3[26716] = {X 393.2861, Y 94.5626, Z -4.6667, A 0.000, B 0.000, C 0.000 }
gfCNCPoint3[26717] = {X 393.9245, Y 93.9287, Z -4.6667, A 0.000, B 0.000, C 0.000 }
gfCNCPoint3[26718] = {X 394.6884, Y 93.4534, Z -4.6667, A 0.000, B 0.000, C 0.000 }
gfCNCPoint3[26719] = {X 395.5393, Y 93.1610, Z -4.6667, A 0.000, B 0.000, C 0.000 }
gfCNCPoint3[26720] = {X 396.4339, Y 93.0660, Z -4.6667, A 0.000, B 0.000, C 0.000 }
gfCNCPoint3[26721] = {X 397.3850, Y 93.0222, Z -4.6667, A 0.000, B 0.000, C 0.000 }
gfCNCPoint3[26722] = {X 398.3327, Y 92.9319, Z -4.6667, A 0.000, B 0.000, C 0.000 }
gfCNCPoint3[26723] = {X 399.0537, Y 92.7571, Z -4.6667, A 0.000, B 0.000, C 0.000 }
gfCNCPoint3[26724] = {X 399.7177, Y 92.4262, Z -4.6667, A 0.000, B 0.000, C 0.000 }
gfCNCPoint3[26725] = {X 405.3922, Y 88.7698, Z -4.6667, A 0.000, B 0.000, C 0.000 }
gfCNCPoint3[26726] = {X 413.9652, Y 83.2880, Z -4.6667, A 0.000, B 0.000, C 0.000 }
gfCNCPoint3[26727] = {X 411.7673, Y 79.8506, Z -4.6667, A 0.000, B 0.000, C 0.000 }
gfCNCPoint3[26728] = {X 411.7673, Y 79.8506, Z -1.6667, A 0.000, B 0.000, C 0.000 }
gfCNCPoint3[26729] = {X 411.7673, Y 79.8506, Z 11.0000, A 0.000, B 0.000, C 0.000 }
gfCNCPoint3[26730] = {X 466.3108, Y 28.5934, Z 11.0000, A 0.000, B 0.000, C 0.000 }
gfCNCPoint3[26731] = {X 466.3108, Y 28.5934, Z -1.6667, A 0.000, B 0.000, C 0.000 }
gfCNCPoint3[26732] = {X 466.3108, Y 28.5934, Z -4.6667, A 0.000, B 0.000, C 0.000 }
gfCNCPoint3[26733] = {X 462.2308, Y 28.5935, Z -4.6667, A 0.000, B 0.000, C 0.000 }
gfCNCPoint3[26734] = {X 462.2310, Y 40.9135, Z -4.6667, A 0.000, B 0.000, C 0.000 }
gfCNCPoint3[26735] = {X 462.2396, Y 40.9205, Z -4.6667, A 0.000, B 0.000, C 0.000 }
gfCNCPoint3[26736] = {X 462.8744, Y 41.5910, Z -4.6667, A 0.000, B 0.000, C 0.000 }
gfCNCPoint3[26737] = {X 463.3522, Y 42.3810, Z -4.6667, A 0.000, B 0.000, C 0.000 }
gfCNCPoint3[26738] = {X 463.6512, Y 43.2546, Z -4.6667, A 0.000, B 0.000, C 0.000 }
gfCNCPoint3[26739] = {X 463.7578, Y 44.1718, Z -4.6667, A 0.000, B 0.000, C 0.000 }
gfCNCPoint3[26740] = {X 463.7579, Y 45.0000, Z -4.6667, A 0.000, B 0.000, C 0.000 }
gfCNCPoint3[26741] = {X 463.6496, Y 45.9613, Z -4.6667, A 0.000, B 0.000, C 0.000 }
gfCNCPoint3[26742] = {X 463.3301, Y 46.8744, Z -4.6667, A 0.000, B 0.000, C 0.000 }
gfCNCPoint3[26743] = {X 462.8155, Y 47.6935, Z -4.6667, A 0.000, B 0.000, C 0.000 }
gfCNCPoint3[26744] = {X 462.1314, Y 48.3775, Z -4.6667, A 0.000, B 0.000, C 0.000 }
gfCNCPoint3[26745] = {X 461.3123, Y 48.8922, Z -4.6667, A 0.000, B 0.000, C 0.000 }
gfCNCPoint3[26746] = {X 460.3992, Y 49.2117, Z -4.6667, A 0.000, B 0.000, C 0.000 }
gfCNCPoint3[26747] = {X 459.4379, Y 49.3200, Z -4.6667, A 0.000, B 0.000, C 0.000 }
gfCNCPoint3[26748] = {X 452.9945, Y 49.3200, Z -4.6667, A 0.000, B 0.000, C 0.000 }
gfCNCPoint3[26749] = {X 452.0380, Y 49.2128, Z -4.6667, A 0.000, B 0.000, C 0.000 }
gfCNCPoint3[26750] = {X 451.1291, Y 48.8965, Z -4.6667, A 0.000, B 0.000, C 0.000 }
gfCNCPoint3[26751] = {X 450.3127, Y 48.3868, Z -4.6667, A 0.000, B 0.000, C 0.000 }
gfCNCPoint3[26752] = {X 449.6294, Y 47.7091, Z -4.6667, A 0.000, B 0.000, C 0.000 }
gfCNCPoint3[26753] = {X 449.1132, Y 46.8968, Z -4.6667, A 0.000, B 0.000, C 0.000 }
gfCNCPoint3[26754] = {X 448.7895, Y 45.9905, Z -4.6667, A 0.000, B 0.000, C 0.000 }
gfCNCPoint3[26755] = {X 448.6746, Y 45.0349, Z -4.6667, A 0.000, B 0.000, C 0.000 }
gfCNCPoint3[26756] = {X 448.6749, Y 44.1494, Z -4.6667, A 0.000, B 0.000, C 0.000 }
gfCNCPoint3[26757] = {X 448.7853, Y 43.2364, Z -4.6667, A 0.000, B 0.000, C 0.000 }
gfCNCPoint3[26758] = {X 449.0865, Y 42.3675, Z -4.6667, A 0.000, B 0.000, C 0.000 }
gfCNCPoint3[26759] = {X 449.5648, Y 41.5821, Z -4.6667, A 0.000, B 0.000, C 0.000 }
gfCNCPoint3[26760] = {X 450.1984, Y 40.9157, Z -4.6667, A 0.000, B 0.000, C 0.000 }
gfCNCPoint3[26761] = {X 450.1984, Y 34.4738, Z -4.6667, A 0.000, B 0.000, C 0.000 }
gfCNCPoint3[26762] = {X 447.4746, Y 34.4738, Z -4.6667, A 0.000, B 0.000, C 0.000 }
gfCNCPoint3[26763] = {X 443.1897, Y 42.8167, Z -4.6667, A 0.000, B 0.000, C 0.000 }
gfCNCPoint3[26764] = {X 443.1946, Y 42.8303, Z -4.6667, A 0.000, B 0.000, C 0.000 }
gfCNCPoint3[26765] = {X 443.3605, Y 43.4914, Z -4.6667, A 0.000, B 0.000, C 0.000 }
gfCNCPoint3[26766] = {X 443.4203, Y 44.1703, Z -4.6667, A 0.000, B 0.000, C 0.000 }
gfCNCPoint3[26767] = {X 443.4205, Y 45.0000, Z -4.6667, A 0.000, B 0.000, C 0.000 }
gfCNCPoint3[26768] = {X 443.3122, Y 45.9613, Z -4.6667, A 0.000, B 0.000, C 0.000 }
gfCNCPoint3[26769] = {X 442.9927, Y 46.8744, Z -4.6667, A 0.000, B 0.000, C 0.000 }
gfCNCPoint3[26770] = {X 442.4780, Y 47.6935, Z -4.6667, A 0.000, B 0.000, C 0.000 }
gfCNCPoint3[26771] = {X 441.7939, Y 48.3775, Z -4.6667, A 0.000, B 0.000, C 0.000 }
gfCNCPoint3[26772] = {X 440.9748, Y 48.8922, Z -4.6667, A 0.000, B 0.000, C 0.000 }
gfCNCPoint3[26773] = {X 440.0618, Y 49.2117, Z -4.6667, A 0.000, B 0.000, C 0.000 }
gfCNCPoint3[26774] = {X 439.1005, Y 49.3200, Z -4.6667, A 0.000, B 0.000, C 0.000 }
gfCNCPoint3[26775] = {X 432.5144, Y 49.3200, Z -4.6667, A 0.000, B 0.000, C 0.000 }
gfCNCPoint3[26776] = {X 431.5531, Y 49.2117, Z -4.6667, A 0.000, B 0.000, C 0.000 }
gfCNCPoint3[26777] = {X 430.6401, Y 48.8922, Z -4.6667, A 0.000, B 0.000, C 0.000 }
gfCNCPoint3[26778] = {X 429.8210, Y 48.3775, Z -4.6667, A 0.000, B 0.000, C 0.000 }
gfCNCPoint3[26779] = {X 429.1369, Y 47.6935, Z -4.6667, A 0.000, B 0.000, C 0.000 }
gfCNCPoint3[26780] = {X 428.6223, Y 46.8745, Z -4.6667, A 0.000, B 0.000, C 0.000 }
gfCNCPoint3[26781] = {X 428.3027, Y 45.9614, Z -4.6667, A 0.000, B 0.000, C 0.000 }
gfCNCPoint3[26782] = {X 428.1944, Y 45.0001, Z -4.6667, A 0.000, B 0.000, C 0.000 }
gfCNCPoint3[26783] = {X 428.1948, Y 44.1494, Z -4.6667, A 0.000, B 0.000, C 0.000 }
gfCNCPoint3[26784] = {X 428.2925, Y 43.2935, Z -4.6667, A 0.000, B 0.000, C 0.000 }
gfCNCPoint3[26785] = {X 428.5580, Y 42.4740, Z -4.6667, A 0.000, B 0.000, C 0.000 }
gfCNCPoint3[26786] = {X 428.9809, Y 41.7236, Z -4.6667, A 0.000, B 0.000, C 0.000 }
gfCNCPoint3[26787] = {X 429.5442, Y 41.0719, Z -4.6667, A 0.000, B 0.000, C 0.000 }
gfCNCPoint3[26788] = {X 430.2256, Y 40.5449, Z -4.6667, A 0.000, B 0.000, C 0.000 }
gfCNCPoint3[26789] = {X 430.9981, Y 40.1637, Z -4.6667, A 0.000, B 0.000, C 0.000 }
gfCNCPoint3[26790] = {X 434.9873, Y 32.3552, Z -4.6667, A 0.000, B 0.000, C 0.000 }
gfCNCPoint3[26791] = {X 433.7210, Y 31.4920, Z -4.6667, A 0.000, B 0.000, C 0.000 }
gfCNCPoint3[26792] = {X 432.5820, Y 30.4665, Z -4.6667, A 0.000, B 0.000, C 0.000 }
gfCNCPoint3[26793] = {X 431.5911, Y 29.2974, Z -4.6667, A 0.000, B 0.000, C 0.000 }
gfCNCPoint3[26794] = {X 430.7662, Y 28.0058, Z -4.6667, A 0.000, B 0.000, C 0.000 }
gfCNCPoint3[26795] = {X 430.1222, Y 26.6152, Z -4.6667, A 0.000, B 0.000, C 0.000 }
gfCNCPoint3[26796] = {X 429.6708, Y 25.1506, Z -4.6667, A 0.000, B 0.000, C 0.000 }
gfCNCPoint3[26797] = {X 429.3569, Y 23.4676, Z -4.6667, A 0.000, B 0.000, C 0.000 }
gfCNCPoint3[26798] = {X 429.2165, Y 21.7613, Z -4.6667, A 0.000, B 0.000, C 0.000 }
gfCNCPoint3[26799] = {X 429.2512, Y 20.0496, Z -4.6667, A 0.000, B 0.000, C 0.000 }
gfCNCPoint3[26800] = {X 429.4607, Y 18.3504, Z -4.6667, A 0.000, B 0.000, C 0.000 }
gfCNCPoint3[26801] = {X 429.8427, Y 16.6815, Z -4.6667, A 0.000, B 0.000, C 0.000 }
gfCNCPoint3[26802] = {X 430.4016, Y 15.1285, Z -4.6667, A 0.000, B 0.000, C 0.000 }
gfCNCPoint3[26803] = {X 431.1714, Y 13.6683, Z -4.6667, A 0.000, B 0.000, C 0.000 }
gfCNCPoint3[26804] = {X 432.1368, Y 12.3296, Z -4.6667, A 0.000, B 0.000, C 0.000 }
gfCNCPoint3[26805] = {X 433.2793, Y 11.1383, Z -4.6667, A 0.000, B 0.000, C 0.000 }
gfCNCPoint3[26806] = {X 434.5764, Y 10.1176, Z -4.6667, A 0.000, B 0.000, C 0.000 }
gfCNCPoint3[26807] = {X 436.0030, Y 9.2874, Z -4.6667, A 0.000, B 0.000, C 0.000 }
gfCNCPoint3[26808] = {X 437.5313, Y 8.6639, Z -4.6667, A 0.000, B 0.000, C 0.000 }
gfCNCPoint3[26809] = {X 439.1315, Y 8.2592, Z -4.6667, A 0.000, B 0.000, C 0.000 }
gfCNCPoint3[26810] = {X 441.2286, Y 7.9686, Z -4.6667, A 0.000, B 0.000, C 0.000 }
gfCNCPoint3[26811] = {X 443.3436, Y 7.8746, Z -4.6667, A 0.000, B 0.000, C 0.000 }
gfCNCPoint3[26812] = {X 444.0357, Y 7.8706, Z -4.6667, A 0.000, B 0.000, C 0.000 }
gfCNCPoint3[26813] = {X 459.4467, Y 7.8706, Z -4.6667, A 0.000, B 0.000, C 0.000 }
gfCNCPoint3[26814] = {X 460.4061, Y 7.9787, Z -4.6667, A 0.000, B 0.000, C 0.000 }
gfCNCPoint3[26815] = {X 461.3173, Y 8.2975, Z -4.6667, A 0.000, B 0.000, C 0.000 }
gfCNCPoint3[26816] = {X 462.1347, Y 8.8111, Z -4.6667, A 0.000, B 0.000, C 0.000 }
gfCNCPoint3[26817] = {X 462.8174, Y 9.4938, Z -4.6667, A 0.000, B 0.000, C 0.000 }
gfCNCPoint3[26818] = {X 463.3310, Y 10.3112, Z -4.6667, A 0.000, B 0.000, C 0.000 }
gfCNCPoint3[26819] = {X 463.6498, Y 11.2225, Z -4.6667, A 0.000, B 0.000, C 0.000 }
gfCNCPoint3[26820] = {X 463.7579, Y 12.1818, Z -4.6667, A 0.000, B 0.000, C 0.000 }
gfCNCPoint3[26821] = {X 463.7579, Y 12.9782, Z -4.6667, A 0.000, B 0.000, C 0.000 }
gfCNCPoint3[26822] = {X 463.6566, Y 13.9080, Z -4.6667, A 0.000, B 0.000, C 0.000 }
gfCNCPoint3[26823] = {X 463.3574, Y 14.7942, Z -4.6667, A 0.000, B 0.000, C 0.000 }
gfCNCPoint3[26824] = {X 462.8746, Y 15.5952, Z -4.6667, A 0.000, B 0.000, C 0.000 }
gfCNCPoint3[26825] = {X 462.2306, Y 16.2735, Z -4.6667, A 0.000, B 0.000, C 0.000 }
gfCNCPoint3[26826] = {X 462.2308, Y 28.5935, Z -4.6667, A 0.000, B 0.000, C 0.000 }
gfCNCPoint3[26827] = {X 466.2308, Y 28.5934, Z -4.6667, A 0.000, B 0.000, C 0.000 }
gfCNCPoint3[26828] = {X 462.1508, Y 28.5935, Z -4.6667, A 0.000, B 0.000, C 0.000 }
gfCNCPoint3[26829] = {X 462.1511, Y 40.9514, Z -4.6667, A 0.000, B 0.000, C 0.000 }
gfCNCPoint3[26830] = {X 462.1884, Y 40.9819, Z -4.6667, A 0.000, B 0.000, C 0.000 }
gfCNCPoint3[26831] = {X 462.8112, Y 41.6399, Z -4.6667, A 0.000, B 0.000, C 0.000 }
gfCNCPoint3[26832] = {X 463.2799, Y 42.4153, Z -4.6667, A 0.000, B 0.000, C 0.000 }
gfCNCPoint3[26833] = {X 463.5733, Y 43.2725, Z -4.6667, A 0.000, B 0.000, C 0.000 }
gfCNCPoint3[26834] = {X 463.6778, Y 44.1724, Z -4.6667, A 0.000, B 0.000, C 0.000 }
gfCNCPoint3[26835] = {X 463.6779, Y 45.0000, Z -4.6667, A 0.000, B 0.000, C 0.000 }
gfCNCPoint3[26836] = {X 463.5716, Y 45.9435, Z -4.6667, A 0.000, B 0.000, C 0.000 }
gfCNCPoint3[26837] = {X 463.2580, Y 46.8397, Z -4.6667, A 0.000, B 0.000, C 0.000 }
gfCNCPoint3[26838] = {X 462.7529, Y 47.6436, Z -4.6667, A 0.000, B 0.000, C 0.000 }
gfCNCPoint3[26839] = {X 462.0815, Y 48.3150, Z -4.6667, A 0.000, B 0.000, C 0.000 }
gfCNCPoint3[26840] = {X 461.2776, Y 48.8201, Z -4.6667, A 0.000, B 0.000, C 0.000 }
gfCNCPoint3[26841] = {X 460.3814, Y 49.1337, Z -4.6667, A 0.000, B 0.000, C 0.000 }
gfCNCPoint3[26842] = {X 459.4379, Y 49.2400, Z -4.6667, A 0.000, B 0.000, C 0.000 }
gfCNCPoint3[26843] = {X 452.9945, Y 49.2400, Z -4.6667, A 0.000, B 0.000, C 0.000 }
gfCNCPoint3[26844] = {X 452.0558, Y 49.1348, Z -4.6667, A 0.000, B 0.000, C 0.000 }
gfCNCPoint3[26845] = {X 451.1636, Y 48.8243, Z -4.6667, A 0.000, B 0.000, C 0.000 }
gfCNCPoint3[26846] = {X 450.3624, Y 48.3241, Z -4.6667, A 0.000, B 0.000, C 0.000 }
gfCNCPoint3[26847] = {X 449.6918, Y 47.6589, Z -4.6667, A 0.000, B 0.000, C 0.000 }
gfCNCPoint3[26848] = {X 449.1851, Y 46.8617, Z -4.6667, A 0.000, B 0.000, C 0.000 }
gfCNCPoint3[26849] = {X 448.8674, Y 45.9721, Z -4.6667, A 0.000, B 0.000, C 0.000 }
gfCNCPoint3[26850] = {X 448.7546, Y 45.0343, Z -4.6667, A 0.000, B 0.000, C 0.000 }
gfCNCPoint3[26851] = {X 448.7549, Y 44.1505, Z -4.6667, A 0.000, B 0.000, C 0.000 }
gfCNCPoint3[26852] = {X 448.8654, Y 43.2454, Z -4.6667, A 0.000, B 0.000, C 0.000 }
gfCNCPoint3[26853] = {X 449.1668, Y 42.3850, Z -4.6667, A 0.000, B 0.000, C 0.000 }
gfCNCPoint3[26854] = {X 449.6452, Y 41.6088, Z -4.6667, A 0.000, B 0.000, C 0.000 }
gfCNCPoint3[26855] = {X 450.2784, Y 40.9529, Z -4.6667, A 0.000, B 0.000, C 0.000 }
gfCNCPoint3[26856] = {X 450.2784, Y 34.3938, Z -4.6667, A 0.000, B 0.000, C 0.000 }
gfCNCPoint3[26857] = {X 447.4258, Y 34.3938, Z -4.6667, A 0.000, B 0.000, C 0.000 }
gfCNCPoint3[26858] = {X 443.1025, Y 42.8113, Z -4.6667, A 0.000, B 0.000, C 0.000 }
gfCNCPoint3[26859] = {X 443.1191, Y 42.8568, Z -4.6667, A 0.000, B 0.000, C 0.000 }
gfCNCPoint3[26860] = {X 443.2817, Y 43.5052, Z -4.6667, A 0.000, B 0.000, C 0.000 }
gfCNCPoint3[26861] = {X 443.3403, Y 44.1710, Z -4.6667, A 0.000, B 0.000, C 0.000 }
gfCNCPoint3[26862] = {X 443.3405, Y 45.0000, Z -4.6667, A 0.000, B 0.000, C 0.000 }
gfCNCPoint3[26863] = {X 443.2342, Y 45.9435, Z -4.6667, A 0.000, B 0.000, C 0.000 }
gfCNCPoint3[26864] = {X 442.9206, Y 46.8397, Z -4.6667, A 0.000, B 0.000, C 0.000 }
gfCNCPoint3[26865] = {X 442.4154, Y 47.6436, Z -4.6667, A 0.000, B 0.000, C 0.000 }
gfCNCPoint3[26866] = {X 441.7441, Y 48.3150, Z -4.6667, A 0.000, B 0.000, C 0.000 }
gfCNCPoint3[26867] = {X 440.9401, Y 48.8201, Z -4.6667, A 0.000, B 0.000, C 0.000 }
gfCNCPoint3[26868] = {X 440.0440, Y 49.1337, Z -4.6667, A 0.000, B 0.000, C 0.000 }
gfCNCPoint3[26869] = {X 439.1005, Y 49.2400, Z -4.6667, A 0.000, B 0.000, C 0.000 }
gfCNCPoint3[26870] = {X 432.5144, Y 49.2400, Z -4.6667, A 0.000, B 0.000, C 0.000 }
gfCNCPoint3[26871] = {X 431.5709, Y 49.1337, Z -4.6667, A 0.000, B 0.000, C 0.000 }
gfCNCPoint3[26872] = {X 430.6748, Y 48.8201, Z -4.6667, A 0.000, B 0.000, C 0.000 }
gfCNCPoint3[26873] = {X 429.8708, Y 48.3150, Z -4.6667, A 0.000, B 0.000, C 0.000 }
gfCNCPoint3[26874] = {X 429.1995, Y 47.6436, Z -4.6667, A 0.000, B 0.000, C 0.000 }
gfCNCPoint3[26875] = {X 428.6943, Y 46.8397, Z -4.6667, A 0.000, B 0.000, C 0.000 }
gfCNCPoint3[26876] = {X 428.3807, Y 45.9436, Z -4.6667, A 0.000, B 0.000, C 0.000 }
gfCNCPoint3[26877] = {X 428.2744, Y 45.0001, Z -4.6667, A 0.000, B 0.000, C 0.000 }
gfCNCPoint3[26878] = {X 428.2748, Y 44.1505, Z -4.6667, A 0.000, B 0.000, C 0.000 }
gfCNCPoint3[26879] = {X 428.3718, Y 43.3054, Z -4.6667, A 0.000, B 0.000, C 0.000 }
gfCNCPoint3[26880] = {X 428.6354, Y 42.4967, Z -4.6667, A 0.000, B 0.000, C 0.000 }
gfCNCPoint3[26881] = {X 429.0552, Y 41.7570, Z -4.6667, A 0.000, B 0.000, C 0.000 }
gfCNCPoint3[26882] = {X 429.6142, Y 41.1159, Z -4.6667, A 0.000, B 0.000, C 0.000 }
gfCNCPoint3[26883] = {X 430.2899, Y 40.5992, Z -4.6667, A 0.000, B 0.000, C 0.000 }
gfCNCPoint3[26884] = {X 431.0551, Y 40.2278, Z -4.6667, A 0.000, B 0.000, C 0.000 }
gfCNCPoint3[26885] = {X 435.0929, Y 32.3242, Z -4.6667, A 0.000, B 0.000, C 0.000 }
gfCNCPoint3[26886] = {X 433.8199, Y 31.4677, Z -4.6667, A 0.000, B 0.000, C 0.000 }
gfCNCPoint3[26887] = {X 432.6745, Y 30.4468, Z -4.6667, A 0.000, B 0.000, C 0.000 }
gfCNCPoint3[26888] = {X 431.6779, Y 29.2802, Z -4.6667, A 0.000, B 0.000, C 0.000 }
gfCNCPoint3[26889] = {X 430.8484, Y 27.9894, Z -4.6667, A 0.000, B 0.000, C 0.000 }
gfCNCPoint3[26890] = {X 430.2014, Y 26.5981, Z -4.6667, A 0.000, B 0.000, C 0.000 }
gfCNCPoint3[26891] = {X 429.7487, Y 25.1321, Z -4.6667, A 0.000, B 0.000, C 0.000 }
gfCNCPoint3[26892] = {X 429.4362, Y 23.4571, Z -4.6667, A 0.000, B 0.000, C 0.000 }
gfCNCPoint3[26893] = {X 429.2964, Y 21.7589, Z -4.6667, A 0.000, B 0.000, C 0.000 }
gfCNCPoint3[26894] = {X 429.3310, Y 20.0553, Z -4.6667, A 0.000, B 0.000, C 0.000 }
gfCNCPoint3[26895] = {X 429.5395, Y 18.3642, Z -4.6667, A 0.000, B 0.000, C 0.000 }
gfCNCPoint3[26896] = {X 429.9196, Y 16.7033, Z -4.6667, A 0.000, B 0.000, C 0.000 }
gfCNCPoint3[26897] = {X 430.4748, Y 15.1607, Z -4.6667, A 0.000, B 0.000, C 0.000 }
gfCNCPoint3[26898] = {X 431.2394, Y 13.7104, Z -4.6667, A 0.000, B 0.000, C 0.000 }
gfCNCPoint3[26899] = {X 432.1984, Y 12.3807, Z -4.6667, A 0.000, B 0.000, C 0.000 }
gfCNCPoint3[26900] = {X 433.3331, Y 11.1974, Z -4.6667, A 0.000, B 0.000, C 0.000 }
gfCNCPoint3[26901] = {X 434.6215, Y 10.1836, Z -4.6667, A 0.000, B 0.000, C 0.000 }
gfCNCPoint3[26902] = {X 436.0385, Y 9.3591, Z -4.6667, A 0.000, B 0.000, C 0.000 }
gfCNCPoint3[26903] = {X 437.5565, Y 8.7398, Z -4.6667, A 0.000, B 0.000, C 0.000 }
gfCNCPoint3[26904] = {X 439.1459, Y 8.3379, Z -4.6667, A 0.000, B 0.000, C 0.000 }
gfCNCPoint3[26905] = {X 441.2359, Y 8.0483, Z -4.6667, A 0.000, B 0.000, C 0.000 }
gfCNCPoint3[26906] = {X 443.3437, Y 7.9546, Z -4.6667, A 0.000, B 0.000, C 0.000 }
gfCNCPoint3[26907] = {X 444.0360, Y 7.9506, Z -4.6667, A 0.000, B 0.000, C 0.000 }
gfCNCPoint3[26908] = {X 459.4467, Y 7.9506, Z -4.6667, A 0.000, B 0.000, C 0.000 }
gfCNCPoint3[26909] = {X 460.3883, Y 8.0567, Z -4.6667, A 0.000, B 0.000, C 0.000 }
gfCNCPoint3[26910] = {X 461.2826, Y 8.3696, Z -4.6667, A 0.000, B 0.000, C 0.000 }
gfCNCPoint3[26911] = {X 462.0848, Y 8.8737, Z -4.6667, A 0.000, B 0.000, C 0.000 }
gfCNCPoint3[26912] = {X 462.7548, Y 9.5437, Z -4.6667, A 0.000, B 0.000, C 0.000 }
gfCNCPoint3[26913] = {X 463.2589, Y 10.3459, Z -4.6667, A 0.000, B 0.000, C 0.000 }
gfCNCPoint3[26914] = {X 463.5719, Y 11.2403, Z -4.6667, A 0.000, B 0.000, C 0.000 }
gfCNCPoint3[26915] = {X 463.6779, Y 12.1818, Z -4.6667, A 0.000, B 0.000, C 0.000 }
gfCNCPoint3[26916] = {X 463.6779, Y 12.9781, Z -4.6667, A 0.000, B 0.000, C 0.000 }
gfCNCPoint3[26917] = {X 463.5764, Y 13.8998, Z -4.6667, A 0.000, B 0.000, C 0.000 }
gfCNCPoint3[26918] = {X 463.2771, Y 14.7773, Z -4.6667, A 0.000, B 0.000, C 0.000 }
gfCNCPoint3[26919] = {X 462.7941, Y 15.5687, Z -4.6667, A 0.000, B 0.000, C 0.000 }
gfCNCPoint3[26920] = {X 462.1506, Y 16.2363, Z -4.6667, A 0.000, B 0.000, C 0.000 }
gfCNCPoint3[26921] = {X 462.1508, Y 28.5935, Z -4.6667, A 0.000, B 0.000, C 0.000 }
gfCNCPoint3[26922] = {X 466.1508, Y 28.5934, Z -4.6667, A 0.000, B 0.000, C 0.000 }
gfCNCPoint3[26923] = {X 462.0708, Y 28.5935, Z -4.6667, A 0.000, B 0.000, C 0.000 }
gfCNCPoint3[26924] = {X 462.0711, Y 40.9894, Z -4.6667, A 0.000, B 0.000, C 0.000 }
gfCNCPoint3[26925] = {X 462.1371, Y 41.0433, Z -4.6667, A 0.000, B 0.000, C 0.000 }
gfCNCPoint3[26926] = {X 462.7479, Y 41.6889, Z -4.6667, A 0.000, B 0.000, C 0.000 }
gfCNCPoint3[26927] = {X 463.2076, Y 42.4495, Z -4.6667, A 0.000, B 0.000, C 0.000 }
gfCNCPoint3[26928] = {X 463.4953, Y 43.2903, Z -4.6667, A 0.000, B 0.000, C 0.000 }
gfCNCPoint3[26929] = {X 463.5978, Y 44.1731, Z -4.6667, A 0.000, B 0.000, C 0.000 }
gfCNCPoint3[26930] = {X 463.5979, Y 45.0000, Z -4.6667, A 0.000, B 0.000, C 0.000 }
gfCNCPoint3[26931] = {X 463.4936, Y 45.9257, Z -4.6667, A 0.000, B 0.000, C 0.000 }
gfCNCPoint3[26932] = {X 463.1860, Y 46.8050, Z -4.6667, A 0.000, B 0.000, C 0.000 }
gfCNCPoint3[26933] = {X 462.6904, Y 47.5937, Z -4.6667, A 0.000, B 0.000, C 0.000 }
gfCNCPoint3[26934] = {X 462.0317, Y 48.2524, Z -4.6667, A 0.000, B 0.000, C 0.000 }
gfCNCPoint3[26935] = {X 461.2429, Y 48.7480, Z -4.6667, A 0.000, B 0.000, C 0.000 }
gfCNCPoint3[26936] = {X 460.3636, Y 49.0557, Z -4.6667, A 0.000, B 0.000, C 0.000 }
gfCNCPoint3[26937] = {X 459.4379, Y 49.1600, Z -4.6667, A 0.000, B 0.000, C 0.000 }
gfCNCPoint3[26938] = {X 452.9945, Y 49.1600, Z -4.6667, A 0.000, B 0.000, C 0.000 }
gfCNCPoint3[26939] = {X 452.0735, Y 49.0568, Z -4.6667, A 0.000, B 0.000, C 0.000 }
gfCNCPoint3[26940] = {X 451.1982, Y 48.7522, Z -4.6667, A 0.000, B 0.000, C 0.000 }
gfCNCPoint3[26941] = {X 450.4120, Y 48.2614, Z -4.6667, A 0.000, B 0.000, C 0.000 }
gfCNCPoint3[26942] = {X 449.7541, Y 47.6087, Z -4.6667, A 0.000, B 0.000, C 0.000 }
gfCNCPoint3[26943] = {X 449.2569, Y 46.8266, Z -4.6667, A 0.000, B 0.000, C 0.000 }
gfCNCPoint3[26944] = {X 448.9453, Y 45.9538, Z -4.6667, A 0.000, B 0.000, C 0.000 }
gfCNCPoint3[26945] = {X 448.8346, Y 45.0336, Z -4.6667, A 0.000, B 0.000, C 0.000 }
gfCNCPoint3[26946] = {X 448.8349, Y 44.1516, Z -4.6667, A 0.000, B 0.000, C 0.000 }
gfCNCPoint3[26947] = {X 448.9454, Y 43.2545, Z -4.6667, A 0.000, B 0.000, C 0.000 }
gfCNCPoint3[26948] = {X 449.2471, Y 42.4026, Z -4.6667, A 0.000, B 0.000, C 0.000 }
gfCNCPoint3[26949] = {X 449.7256, Y 41.6358, Z -4.6667, A 0.000, B 0.000, C 0.000 }
gfCNCPoint3[26950] = {X 450.3584, Y 40.9906, Z -4.6667, A 0.000, B 0.000, C 0.000 }
gfCNCPoint3[26951] = {X 450.3584, Y 34.3138, Z -4.6667, A 0.000, B 0.000, C 0.000 }
gfCNCPoint3[26952] = {X 447.3769, Y 34.3138, Z -4.6667, A 0.000, B 0.000, C 0.000 }
gfCNCPoint3[26953] = {X 443.0153, Y 42.8059, Z -4.6667, A 0.000, B 0.000, C 0.000 }
gfCNCPoint3[26954] = {X 443.0436, Y 42.8833, Z -4.6667, A 0.000, B 0.000, C 0.000 }
gfCNCPoint3[26955] = {X 443.2029, Y 43.5190, Z -4.6667, A 0.000, B 0.000, C 0.000 }
gfCNCPoint3[26956] = {X 443.2603, Y 44.1717, Z -4.6667, A 0.000, B 0.000, C 0.000 }
gfCNCPoint3[26957] = {X 443.2605, Y 45.0000, Z -4.6667, A 0.000, B 0.000, C 0.000 }
gfCNCPoint3[26958] = {X 443.1562, Y 45.9257, Z -4.6667, A 0.000, B 0.000, C 0.000 }
gfCNCPoint3[26959] = {X 442.8485, Y 46.8050, Z -4.6667, A 0.000, B 0.000, C 0.000 }
gfCNCPoint3[26960] = {X 442.3529, Y 47.5937, Z -4.6667, A 0.000, B 0.000, C 0.000 }
gfCNCPoint3[26961] = {X 441.6942, Y 48.2524, Z -4.6667, A 0.000, B 0.000, C 0.000 }
gfCNCPoint3[26962] = {X 440.9054, Y 48.7480, Z -4.6667, A 0.000, B 0.000, C 0.000 }
gfCNCPoint3[26963] = {X 440.0262, Y 49.0557, Z -4.6667, A 0.000, B 0.000, C 0.000 }
gfCNCPoint3[26964] = {X 439.1005, Y 49.1600, Z -4.6667, A 0.000, B 0.000, C 0.000 }
gfCNCPoint3[26965] = {X 432.5144, Y 49.1600, Z -4.6667, A 0.000, B 0.000, C 0.000 }
gfCNCPoint3[26966] = {X 431.5887, Y 49.0557, Z -4.6667, A 0.000, B 0.000, C 0.000 }
gfCNCPoint3[26967] = {X 430.7095, Y 48.7480, Z -4.6667, A 0.000, B 0.000, C 0.000 }
gfCNCPoint3[26968] = {X 429.9207, Y 48.2524, Z -4.6667, A 0.000, B 0.000, C 0.000 }
gfCNCPoint3[26969] = {X 429.2620, Y 47.5937, Z -4.6667, A 0.000, B 0.000, C 0.000 }
gfCNCPoint3[26970] = {X 428.7664, Y 46.8050, Z -4.6667, A 0.000, B 0.000, C 0.000 }
gfCNCPoint3[26971] = {X 428.4587, Y 45.9257, Z -4.6667, A 0.000, B 0.000, C 0.000 }
gfCNCPoint3[26972] = {X 428.3544, Y 45.0000, Z -4.6667, A 0.000, B 0.000, C 0.000 }
gfCNCPoint3[26973] = {X 428.3548, Y 44.1516, Z -4.6667, A 0.000, B 0.000, C 0.000 }
gfCNCPoint3[26974] = {X 428.4510, Y 43.3174, Z -4.6667, A 0.000, B 0.000, C 0.000 }
gfCNCPoint3[26975] = {X 428.7128, Y 42.5195, Z -4.6667, A 0.000, B 0.000, C 0.000 }
gfCNCPoint3[26976] = {X 429.1295, Y 41.7905, Z -4.6667, A 0.000, B 0.000, C 0.000 }
gfCNCPoint3[26977] = {X 429.6841, Y 41.1600, Z -4.6667, A 0.000, B 0.000, C 0.000 }
gfCNCPoint3[26978] = {X 430.3541, Y 40.6537, Z -4.6667, A 0.000, B 0.000, C 0.000 }
gfCNCPoint3[26979] = {X 431.1120, Y 40.2923, Z -4.6667, A 0.000, B 0.000, C 0.000 }
gfCNCPoint3[26980] = {X 435.1989, Y 32.2927, Z -4.6667, A 0.000, B 0.000, C 0.000 }
gfCNCPoint3[26981] = {X 433.9190, Y 31.4432, Z -4.6667, A 0.000, B 0.000, C 0.000 }
gfCNCPoint3[26982] = {X 432.7671, Y 30.4269, Z -4.6667, A 0.000, B 0.000, C 0.000 }
gfCNCPoint3[26983] = {X 431.7648, Y 29.2628, Z -4.6667, A 0.000, B 0.000, C 0.000 }
gfCNCPoint3[26984] = {X 430.9307, Y 27.9728, Z -4.6667, A 0.000, B 0.000, C 0.000 }
gfCNCPoint3[26985] = {X 430.2805, Y 26.5810, Z -4.6667, A 0.000, B 0.000, C 0.000 }
gfCNCPoint3[26986] = {X 429.8265, Y 25.1135, Z -4.6667, A 0.000, B 0.000, C 0.000 }
gfCNCPoint3[26987] = {X 429.5155, Y 23.4466, Z -4.6667, A 0.000, B 0.000, C 0.000 }
gfCNCPoint3[26988] = {X 429.3764, Y 21.7565, Z -4.6667, A 0.000, B 0.000, C 0.000 }
gfCNCPoint3[26989] = {X 429.4108, Y 20.0611, Z -4.6667, A 0.000, B 0.000, C 0.000 }
gfCNCPoint3[26990] = {X 429.6183, Y 18.3781, Z -4.6667, A 0.000, B 0.000, C 0.000 }
gfCNCPoint3[26991] = {X 429.9966, Y 16.7251, Z -4.6667, A 0.000, B 0.000, C 0.000 }
gfCNCPoint3[26992] = {X 430.5480, Y 15.1930, Z -4.6667, A 0.000, B 0.000, C 0.000 }
gfCNCPoint3[26993] = {X 431.3074, Y 13.7526, Z -4.6667, A 0.000, B 0.000, C 0.000 }
gfCNCPoint3[26994] = {X 432.2599, Y 12.4319, Z -4.6667, A 0.000, B 0.000, C 0.000 }
gfCNCPoint3[26995] = {X 433.3869, Y 11.2566, Z -4.6667, A 0.000, B 0.000, C 0.000 }
gfCNCPoint3[26996] = {X 434.6666, Y 10.2497, Z -4.6667, A 0.000, B 0.000, C 0.000 }
gfCNCPoint3[26997] = {X 436.0740, Y 9.4308, Z -4.6667, A 0.000, B 0.000, C 0.000 }
gfCNCPoint3[26998] = {X 437.5817, Y 8.8157, Z -4.6667, A 0.000, B 0.000, C 0.000 }
gfCNCPoint3[26999] = {X 439.1604, Y 8.4165, Z -4.6667, A 0.000, B 0.000, C 0.000 }
gfCNCPoint3[27000] = {X 441.2432, Y 8.1280, Z -4.6667, A 0.000, B 0.000, C 0.000 }
gfCNCPoint3[27001] = {X 443.3439, Y 8.0346, Z -4.6667, A 0.000, B 0.000, C 0.000 }
gfCNCPoint3[27002] = {X 444.0362, Y 8.0306, Z -4.6667, A 0.000, B 0.000, C 0.000 }
gfCNCPoint3[27003] = {X 459.4467, Y 8.0306, Z -4.6667, A 0.000, B 0.000, C 0.000 }
gfCNCPoint3[27004] = {X 460.3705, Y 8.1346, Z -4.6667, A 0.000, B 0.000, C 0.000 }
gfCNCPoint3[27005] = {X 461.2479, Y 8.4417, Z -4.6667, A 0.000, B 0.000, C 0.000 }
gfCNCPoint3[27006] = {X 462.0350, Y 8.9362, Z -4.6667, A 0.000, B 0.000, C 0.000 }
gfCNCPoint3[27007] = {X 462.6923, Y 9.5935, Z -4.6667, A 0.000, B 0.000, C 0.000 }
gfCNCPoint3[27008] = {X 463.1868, Y 10.3806, Z -4.6667, A 0.000, B 0.000, C 0.000 }
gfCNCPoint3[27009] = {X 463.4939, Y 11.2581, Z -4.6667, A 0.000, B 0.000, C 0.000 }
gfCNCPoint3[27010] = {X 463.5979, Y 12.1818, Z -4.6667, A 0.000, B 0.000, C 0.000 }
gfCNCPoint3[27011] = {X 463.5979, Y 12.9781, Z -4.6667, A 0.000, B 0.000, C 0.000 }
gfCNCPoint3[27012] = {X 463.5023, Y 13.8651, Z -4.6667, A 0.000, B 0.000, C 0.000 }
gfCNCPoint3[27013] = {X 463.2197, Y 14.7112, Z -4.6667, A 0.000, B 0.000, C 0.000 }
gfCNCPoint3[27014] = {X 462.7632, Y 15.4777, Z -4.6667, A 0.000, B 0.000, C 0.000 }
gfCNCPoint3[27015] = {X 462.1538, Y 16.1292, Z -4.6667, A 0.000, B 0.000, C 0.000 }
gfCNCPoint3[27016] = {X 462.0706, Y 16.1990, Z -4.6667, A 0.000, B 0.000, C 0.000 }
gfCNCPoint3[27017] = {X 462.0708, Y 28.5935, Z -4.6667, A 0.000, B 0.000, C 0.000 }
gfCNCPoint3[27018] = {X 466.0708, Y 28.5935, Z -4.6667, A 0.000, B 0.000, C 0.000 }
gfCNCPoint3[27019] = {X 461.9908, Y 28.5935, Z -4.6667, A 0.000, B 0.000, C 0.000 }
gfCNCPoint3[27020] = {X 461.9911, Y 41.0274, Z -4.6667, A 0.000, B 0.000, C 0.000 }
gfCNCPoint3[27021] = {X 462.0859, Y 41.1048, Z -4.6667, A 0.000, B 0.000, C 0.000 }
gfCNCPoint3[27022] = {X 462.6846, Y 41.7379, Z -4.6667, A 0.000, B 0.000, C 0.000 }
gfCNCPoint3[27023] = {X 463.1353, Y 42.4837, Z -4.6667, A 0.000, B 0.000, C 0.000 }
gfCNCPoint3[27024] = {X 463.4173, Y 43.3082, Z -4.6667, A 0.000, B 0.000, C 0.000 }
gfCNCPoint3[27025] = {X 463.5178, Y 44.1738, Z -4.6667, A 0.000, B 0.000, C 0.000 }
gfCNCPoint3[27026] = {X 463.5179, Y 45.0000, Z -4.6667, A 0.000, B 0.000, C 0.000 }
gfCNCPoint3[27027] = {X 463.4156, Y 45.9079, Z -4.6667, A 0.000, B 0.000, C 0.000 }
gfCNCPoint3[27028] = {X 463.1139, Y 46.7702, Z -4.6667, A 0.000, B 0.000, C 0.000 }
gfCNCPoint3[27029] = {X 462.6278, Y 47.5438, Z -4.6667, A 0.000, B 0.000, C 0.000 }
gfCNCPoint3[27030] = {X 461.9818, Y 48.1899, Z -4.6667, A 0.000, B 0.000, C 0.000 }
gfCNCPoint3[27031] = {X 461.2082, Y 48.6760, Z -4.6667, A 0.000, B 0.000, C 0.000 }
gfCNCPoint3[27032] = {X 460.3458, Y 48.9777, Z -4.6667, A 0.000, B 0.000, C 0.000 }
gfCNCPoint3[27033] = {X 459.4379, Y 49.0800, Z -4.6667, A 0.000, B 0.000, C 0.000 }
gfCNCPoint3[27034] = {X 452.9945, Y 49.0800, Z -4.6667, A 0.000, B 0.000, C 0.000 }
gfCNCPoint3[27035] = {X 452.0912, Y 48.9788, Z -4.6667, A 0.000, B 0.000, C 0.000 }
gfCNCPoint3[27036] = {X 451.2327, Y 48.6800, Z -4.6667, A 0.000, B 0.000, C 0.000 }
gfCNCPoint3[27037] = {X 450.4617, Y 48.1987, Z -4.6667, A 0.000, B 0.000, C 0.000 }
gfCNCPoint3[27038] = {X 449.8164, Y 47.5585, Z -4.6667, A 0.000, B 0.000, C 0.000 }
gfCNCPoint3[27039] = {X 449.3288, Y 46.7914, Z -4.6667, A 0.000, B 0.000, C 0.000 }
gfCNCPoint3[27040] = {X 449.0232, Y 45.9354, Z -4.6667, A 0.000, B 0.000, C 0.000 }
gfCNCPoint3[27041] = {X 448.9146, Y 45.0330, Z -4.6667, A 0.000, B 0.000, C 0.000 }
gfCNCPoint3[27042] = {X 448.9149, Y 44.1527, Z -4.6667, A 0.000, B 0.000, C 0.000 }
gfCNCPoint3[27043] = {X 449.0254, Y 43.2637, Z -4.6667, A 0.000, B 0.000, C 0.000 }
gfCNCPoint3[27044] = {X 449.3274, Y 42.4203, Z -4.6667, A 0.000, B 0.000, C 0.000 }
gfCNCPoint3[27045] = {X 449.8061, Y 41.6631, Z -4.6667, A 0.000, B 0.000, C 0.000 }
gfCNCPoint3[27046] = {X 450.4384, Y 41.0287, Z -4.6667, A 0.000, B 0.000, C 0.000 }
gfCNCPoint3[27047] = {X 450.4384, Y 34.2338, Z -4.6667, A 0.000, B 0.000, C 0.000 }
gfCNCPoint3[27048] = {X 447.3281, Y 34.2338, Z -4.6667, A 0.000, B 0.000, C 0.000 }
gfCNCPoint3[27049] = {X 442.9282, Y 42.8005, Z -4.6667, A 0.000, B 0.000, C 0.000 }
gfCNCPoint3[27050] = {X 442.9681, Y 42.9098, Z -4.6667, A 0.000, B 0.000, C 0.000 }
gfCNCPoint3[27051] = {X 443.1241, Y 43.5327, Z -4.6667, A 0.000, B 0.000, C 0.000 }
gfCNCPoint3[27052] = {X 443.1803, Y 44.1725, Z -4.6667, A 0.000, B 0.000, C 0.000 }
gfCNCPoint3[27053] = {X 443.1805, Y 45.0000, Z -4.6667, A 0.000, B 0.000, C 0.000 }
gfCNCPoint3[27054] = {X 443.0782, Y 45.9079, Z -4.6667, A 0.000, B 0.000, C 0.000 }
gfCNCPoint3[27055] = {X 442.7764, Y 46.7702, Z -4.6667, A 0.000, B 0.000, C 0.000 }
gfCNCPoint3[27056] = {X 442.2903, Y 47.5438, Z -4.6667, A 0.000, B 0.000, C 0.000 }
gfCNCPoint3[27057] = {X 441.6443, Y 48.1899, Z -4.6667, A 0.000, B 0.000, C 0.000 }
gfCNCPoint3[27058] = {X 440.8707, Y 48.6760, Z -4.6667, A 0.000, B 0.000, C 0.000 }
gfCNCPoint3[27059] = {X 440.0084, Y 48.9777, Z -4.6667, A 0.000, B 0.000, C 0.000 }
gfCNCPoint3[27060] = {X 439.1005, Y 49.0800, Z -4.6667, A 0.000, B 0.000, C 0.000 }
gfCNCPoint3[27061] = {X 432.5144, Y 49.0800, Z -4.6667, A 0.000, B 0.000, C 0.000 }
gfCNCPoint3[27062] = {X 431.6065, Y 48.9777, Z -4.6667, A 0.000, B 0.000, C 0.000 }
gfCNCPoint3[27063] = {X 430.7442, Y 48.6760, Z -4.6667, A 0.000, B 0.000, C 0.000 }
gfCNCPoint3[27064] = {X 429.9706, Y 48.1899, Z -4.6667, A 0.000, B 0.000, C 0.000 }
gfCNCPoint3[27065] = {X 429.3245, Y 47.5438, Z -4.6667, A 0.000, B 0.000, C 0.000 }
gfCNCPoint3[27066] = {X 428.8385, Y 46.7702, Z -4.6667, A 0.000, B 0.000, C 0.000 }
gfCNCPoint3[27067] = {X 428.5367, Y 45.9079, Z -4.6667, A 0.000, B 0.000, C 0.000 }
gfCNCPoint3[27068] = {X 428.4344, Y 45.0000, Z -4.6667, A 0.000, B 0.000, C 0.000 }
gfCNCPoint3[27069] = {X 428.4348, Y 44.1527, Z -4.6667, A 0.000, B 0.000, C 0.000 }
gfCNCPoint3[27070] = {X 428.5303, Y 43.3294, Z -4.6667, A 0.000, B 0.000, C 0.000 }
gfCNCPoint3[27071] = {X 428.7902, Y 42.5424, Z -4.6667, A 0.000, B 0.000, C 0.000 }
gfCNCPoint3[27072] = {X 429.2038, Y 41.8242, Z -4.6667, A 0.000, B 0.000, C 0.000 }
gfCNCPoint3[27073] = {X 429.7540, Y 41.2044, Z -4.6667, A 0.000, B 0.000, C 0.000 }
gfCNCPoint3[27074] = {X 430.4181, Y 40.7085, Z -4.6667, A 0.000, B 0.000, C 0.000 }
gfCNCPoint3[27075] = {X 431.1687, Y 40.3571, Z -4.6667, A 0.000, B 0.000, C 0.000 }
gfCNCPoint3[27076] = {X 435.3050, Y 32.2608, Z -4.6667, A 0.000, B 0.000, C 0.000 }
gfCNCPoint3[27077] = {X 434.0183, Y 31.4183, Z -4.6667, A 0.000, B 0.000, C 0.000 }
gfCNCPoint3[27078] = {X 432.8599, Y 30.4068, Z -4.6667, A 0.000, B 0.000, C 0.000 }
gfCNCPoint3[27079] = {X 431.8517, Y 29.2454, Z -4.6667, A 0.000, B 0.000, C 0.000 }
gfCNCPoint3[27080] = {X 431.0130, Y 27.9563, Z -4.6667, A 0.000, B 0.000, C 0.000 }
gfCNCPoint3[27081] = {X 430.3597, Y 26.5640, Z -4.6667, A 0.000, B 0.000, C 0.000 }
gfCNCPoint3[27082] = {X 429.9043, Y 25.0950, Z -4.6667, A 0.000, B 0.000, C 0.000 }
gfCNCPoint3[27083] = {X 429.5948, Y 23.4361, Z -4.6667, A 0.000, B 0.000, C 0.000 }
gfCNCPoint3[27084] = {X 429.4564, Y 21.7542, Z -4.6667, A 0.000, B 0.000, C 0.000 }
gfCNCPoint3[27085] = {X 429.4906, Y 20.0669, Z -4.6667, A 0.000, B 0.000, C 0.000 }
gfCNCPoint3[27086] = {X 429.6970, Y 18.3920, Z -4.6667, A 0.000, B 0.000, C 0.000 }
gfCNCPoint3[27087] = {X 430.0736, Y 16.7469, Z -4.6667, A 0.000, B 0.000, C 0.000 }
gfCNCPoint3[27088] = {X 430.6212, Y 15.2253, Z -4.6667, A 0.000, B 0.000, C 0.000 }
gfCNCPoint3[27089] = {X 431.3754, Y 13.7947, Z -4.6667, A 0.000, B 0.000, C 0.000 }
gfCNCPoint3[27090] = {X 432.3214, Y 12.4830, Z -4.6667, A 0.000, B 0.000, C 0.000 }
gfCNCPoint3[27091] = {X 433.4408, Y 11.3158, Z -4.6667, A 0.000, B 0.000, C 0.000 }
gfCNCPoint3[27092] = {X 434.7117, Y 10.3158, Z -4.6667, A 0.000, B 0.000, C 0.000 }
gfCNCPoint3[27093] = {X 436.1095, Y 9.5025, Z -4.6667, A 0.000, B 0.000, C 0.000 }
gfCNCPoint3[27094] = {X 437.6070, Y 8.8916, Z -4.6667, A 0.000, B 0.000, C 0.000 }
gfCNCPoint3[27095] = {X 439.1748, Y 8.4952, Z -4.6667, A 0.000, B 0.000, C 0.000 }
gfCNCPoint3[27096] = {X 441.2505, Y 8.2076, Z -4.6667, A 0.000, B 0.000, C 0.000 }
gfCNCPoint3[27097] = {X 443.3440, Y 8.1146, Z -4.6667, A 0.000, B 0.000, C 0.000 }
gfCNCPoint3[27098] = {X 444.0364, Y 8.1106, Z -4.6667, A 0.000, B 0.000, C 0.000 }
gfCNCPoint3[27099] = {X 459.4467, Y 8.1106, Z -4.6667, A 0.000, B 0.000, C 0.000 }
gfCNCPoint3[27100] = {X 460.3527, Y 8.2126, Z -4.6667, A 0.000, B 0.000, C 0.000 }
gfCNCPoint3[27101] = {X 461.2132, Y 8.5137, Z -4.6667, A 0.000, B 0.000, C 0.000 }
gfCNCPoint3[27102] = {X 461.9851, Y 8.9988, Z -4.6667, A 0.000, B 0.000, C 0.000 }
gfCNCPoint3[27103] = {X 462.6297, Y 9.6434, Z -4.6667, A 0.000, B 0.000, C 0.000 }
gfCNCPoint3[27104] = {X 463.1148, Y 10.4154, Z -4.6667, A 0.000, B 0.000, C 0.000 }
gfCNCPoint3[27105] = {X 463.4159, Y 11.2759, Z -4.6667, A 0.000, B 0.000, C 0.000 }
gfCNCPoint3[27106] = {X 463.5179, Y 12.1818, Z -4.6667, A 0.000, B 0.000, C 0.000 }
gfCNCPoint3[27107] = {X 463.5179, Y 12.9781, Z -4.6667, A 0.000, B 0.000, C 0.000 }
gfCNCPoint3[27108] = {X 463.4241, Y 13.8480, Z -4.6667, A 0.000, B 0.000, C 0.000 }
gfCNCPoint3[27109] = {X 463.1470, Y 14.6779, Z -4.6667, A 0.000, B 0.000, C 0.000 }
gfCNCPoint3[27110] = {X 462.6993, Y 15.4296, Z -4.6667, A 0.000, B 0.000, C 0.000 }
gfCNCPoint3[27111] = {X 462.1016, Y 16.0686, Z -4.6667, A 0.000, B 0.000, C 0.000 }
gfCNCPoint3[27112] = {X 462.0441, Y 16.1172, Z -4.6667, A 0.000, B 0.000, C 0.000 }
gfCNCPoint3[27113] = {X 461.9858, Y 16.1647, Z -4.6667, A 0.000, B 0.000, C 0.000 }
gfCNCPoint3[27114] = {X 461.9906, Y 16.1990, Z -4.6667, A 0.000, B 0.000, C 0.000 }
gfCNCPoint3[27115] = {X 461.9908, Y 28.5935, Z -4.6667, A 0.000, B 0.000, C 0.000 }
gfCNCPoint3[27116] = {X 465.9908, Y 28.5935, Z -4.6667, A 0.000, B 0.000, C 0.000 }
gfCNCPoint3[27117] = {X 465.9908, Y 28.5933, Z -4.6667, A 0.000, B 0.000, C 0.000 }
gfCNCPoint3[27118] = {X 461.9105, Y 28.5935, Z -4.6667, A 0.000, B 0.000, C 0.000 }
gfCNCPoint3[27119] = {X 461.9111, Y 41.0653, Z -4.6667, A 0.000, B 0.000, C 0.000 }
gfCNCPoint3[27120] = {X 462.0499, Y 41.1793, Z -4.6667, A 0.000, B 0.000, C 0.000 }
gfCNCPoint3[27121] = {X 462.6356, Y 41.8057, Z -4.6667, A 0.000, B 0.000, C 0.000 }
gfCNCPoint3[27122] = {X 463.0744, Y 42.5426, Z -4.6667, A 0.000, B 0.000, C 0.000 }
gfCNCPoint3[27123] = {X 463.3460, Y 43.3562, Z -4.6667, A 0.000, B 0.000, C 0.000 }
gfCNCPoint3[27124] = {X 463.4379, Y 44.2089, Z -4.6667, A 0.000, B 0.000, C 0.000 }
gfCNCPoint3[27125] = {X 463.4379, Y 45.0000, Z -4.6667, A 0.000, B 0.000, C 0.000 }
gfCNCPoint3[27126] = {X 463.3377, Y 45.8901, Z -4.6667, A 0.000, B 0.000, C 0.000 }
gfCNCPoint3[27127] = {X 463.0418, Y 46.7355, Z -4.6667, A 0.000, B 0.000, C 0.000 }
gfCNCPoint3[27128] = {X 462.5653, Y 47.4940, Z -4.6667, A 0.000, B 0.000, C 0.000 }
gfCNCPoint3[27129] = {X 461.9319, Y 48.1273, Z -4.6667, A 0.000, B 0.000, C 0.000 }
gfCNCPoint3[27130] = {X 461.1735, Y 48.6039, Z -4.6667, A 0.000, B 0.000, C 0.000 }
gfCNCPoint3[27131] = {X 460.3280, Y 48.8997, Z -4.6667, A 0.000, B 0.000, C 0.000 }
gfCNCPoint3[27132] = {X 459.4379, Y 49.0000, Z -4.6667, A 0.000, B 0.000, C 0.000 }
gfCNCPoint3[27133] = {X 452.9945, Y 49.0000, Z -4.6667, A 0.000, B 0.000, C 0.000 }
gfCNCPoint3[27134] = {X 452.1044, Y 48.8997, Z -4.6667, A 0.000, B 0.000, C 0.000 }
gfCNCPoint3[27135] = {X 451.2589, Y 48.6039, Z -4.6667, A 0.000, B 0.000, C 0.000 }
gfCNCPoint3[27136] = {X 450.5005, Y 48.1273, Z -4.6667, A 0.000, B 0.000, C 0.000 }
gfCNCPoint3[27137] = {X 449.8671, Y 47.4939, Z -4.6667, A 0.000, B 0.000, C 0.000 }
gfCNCPoint3[27138] = {X 449.3906, Y 46.7355, Z -4.6667, A 0.000, B 0.000, C 0.000 }
gfCNCPoint3[27139] = {X 449.0948, Y 45.8901, Z -4.6667, A 0.000, B 0.000, C 0.000 }
gfCNCPoint3[27140] = {X 448.9945, Y 45.0000, Z -4.6667, A 0.000, B 0.000, C 0.000 }
gfCNCPoint3[27141] = {X 448.9949, Y 44.1538, Z -4.6667, A 0.000, B 0.000, C 0.000 }
gfCNCPoint3[27142] = {X 449.1055, Y 43.2730, Z -4.6667, A 0.000, B 0.000, C 0.000 }
gfCNCPoint3[27143] = {X 449.4077, Y 42.4382, Z -4.6667, A 0.000, B 0.000, C 0.000 }
gfCNCPoint3[27144] = {X 449.8865, Y 41.6907, Z -4.6667, A 0.000, B 0.000, C 0.000 }
gfCNCPoint3[27145] = {X 450.5184, Y 41.0672, Z -4.6667, A 0.000, B 0.000, C 0.000 }
gfCNCPoint3[27146] = {X 450.5184, Y 34.1538, Z -4.6667, A 0.000, B 0.000, C 0.000 }
gfCNCPoint3[27147] = {X 447.5235, Y 34.1538, Z -4.6667, A 0.000, B 0.000, C 0.000 }
gfCNCPoint3[27148] = {X 447.2796, Y 34.1532, Z -4.6667, A 0.000, B 0.000, C 0.000 }
gfCNCPoint3[27149] = {X 443.4077, Y 41.6922, Z -4.6667, A 0.000, B 0.000, C 0.000 }
gfCNCPoint3[27150] = {X 442.8410, Y 42.7951, Z -4.6667, A 0.000, B 0.000, C 0.000 }
gfCNCPoint3[27151] = {X 442.8968, Y 42.9488, Z -4.6667, A 0.000, B 0.000, C 0.000 }
gfCNCPoint3[27152] = {X 443.0492, Y 43.5707, Z -4.6667, A 0.000, B 0.000, C 0.000 }
gfCNCPoint3[27153] = {X 443.1005, Y 44.2089, Z -4.6667, A 0.000, B 0.000, C 0.000 }
gfCNCPoint3[27154] = {X 443.1005, Y 45.0000, Z -4.6667, A 0.000, B 0.000, C 0.000 }
gfCNCPoint3[27155] = {X 443.0002, Y 45.8901, Z -4.6667, A 0.000, B 0.000, C 0.000 }
gfCNCPoint3[27156] = {X 442.7043, Y 46.7355, Z -4.6667, A 0.000, B 0.000, C 0.000 }
gfCNCPoint3[27157] = {X 442.2278, Y 47.4940, Z -4.6667, A 0.000, B 0.000, C 0.000 }
gfCNCPoint3[27158] = {X 441.5944, Y 48.1273, Z -4.6667, A 0.000, B 0.000, C 0.000 }
gfCNCPoint3[27159] = {X 440.8360, Y 48.6039, Z -4.6667, A 0.000, B 0.000, C 0.000 }
gfCNCPoint3[27160] = {X 439.9906, Y 48.8997, Z -4.6667, A 0.000, B 0.000, C 0.000 }
gfCNCPoint3[27161] = {X 439.1005, Y 49.0000, Z -4.6667, A 0.000, B 0.000, C 0.000 }
gfCNCPoint3[27162] = {X 432.5144, Y 49.0000, Z -4.6667, A 0.000, B 0.000, C 0.000 }
gfCNCPoint3[27163] = {X 431.6243, Y 48.8997, Z -4.6667, A 0.000, B 0.000, C 0.000 }
gfCNCPoint3[27164] = {X 430.7789, Y 48.6039, Z -4.6667, A 0.000, B 0.000, C 0.000 }
gfCNCPoint3[27165] = {X 430.0204, Y 48.1273, Z -4.6667, A 0.000, B 0.000, C 0.000 }
gfCNCPoint3[27166] = {X 429.3871, Y 47.4940, Z -4.6667, A 0.000, B 0.000, C 0.000 }
gfCNCPoint3[27167] = {X 428.9105, Y 46.7355, Z -4.6667, A 0.000, B 0.000, C 0.000 }
gfCNCPoint3[27168] = {X 428.6147, Y 45.8901, Z -4.6667, A 0.000, B 0.000, C 0.000 }
gfCNCPoint3[27169] = {X 428.5144, Y 45.0000, Z -4.6667, A 0.000, B 0.000, C 0.000 }
gfCNCPoint3[27170] = {X 428.5148, Y 44.1538, Z -4.6667, A 0.000, B 0.000, C 0.000 }
gfCNCPoint3[27171] = {X 428.6096, Y 43.3414, Z -4.6667, A 0.000, B 0.000, C 0.000 }
gfCNCPoint3[27172] = {X 428.8676, Y 42.5654, Z -4.6667, A 0.000, B 0.000, C 0.000 }
gfCNCPoint3[27173] = {X 429.2781, Y 41.8580, Z -4.6667, A 0.000, B 0.000, C 0.000 }
gfCNCPoint3[27174] = {X 429.8239, Y 41.2489, Z -4.6667, A 0.000, B 0.000, C 0.000 }
gfCNCPoint3[27175] = {X 430.4821, Y 40.7635, Z -4.6667, A 0.000, B 0.000, C 0.000 }
gfCNCPoint3[27176] = {X 431.2253, Y 40.4222, Z -4.6667, A 0.000, B 0.000, C 0.000 }
gfCNCPoint3[27177] = {X 435.4114, Y 32.2284, Z -4.6667, A 0.000, B 0.000, C 0.000 }
gfCNCPoint3[27178] = {X 434.1179, Y 31.3932, Z -4.6667, A 0.000, B 0.000, C 0.000 }
gfCNCPoint3[27179] = {X 432.9528, Y 30.3865, Z -4.6667, A 0.000, B 0.000, C 0.000 }
gfCNCPoint3[27180] = {X 431.9388, Y 29.2279, Z -4.6667, A 0.000, B 0.000, C 0.000 }
gfCNCPoint3[27181] = {X 431.0954, Y 27.9397, Z -4.6667, A 0.000, B 0.000, C 0.000 }
gfCNCPoint3[27182] = {X 430.4389, Y 26.5470, Z -4.6667, A 0.000, B 0.000, C 0.000 }
gfCNCPoint3[27183] = {X 429.9822, Y 25.0766, Z -4.6667, A 0.000, B 0.000, C 0.000 }
gfCNCPoint3[27184] = {X 429.6741, Y 23.4256, Z -4.6667, A 0.000, B 0.000, C 0.000 }
gfCNCPoint3[27185] = {X 429.5363, Y 21.7518, Z -4.6667, A 0.000, B 0.000, C 0.000 }
gfCNCPoint3[27186] = {X 429.5704, Y 20.0727, Z -4.6667, A 0.000, B 0.000, C 0.000 }
gfCNCPoint3[27187] = {X 429.7758, Y 18.4059, Z -4.6667, A 0.000, B 0.000, C 0.000 }
gfCNCPoint3[27188] = {X 430.1505, Y 16.7687, Z -4.6667, A 0.000, B 0.000, C 0.000 }
gfCNCPoint3[27189] = {X 430.6944, Y 15.2576, Z -4.6667, A 0.000, B 0.000, C 0.000 }
gfCNCPoint3[27190] = {X 431.4434, Y 13.8368, Z -4.6667, A 0.000, B 0.000, C 0.000 }
gfCNCPoint3[27191] = {X 432.3829, Y 12.5342, Z -4.6667, A 0.000, B 0.000, C 0.000 }
gfCNCPoint3[27192] = {X 433.4946, Y 11.3750, Z -4.6667, A 0.000, B 0.000, C 0.000 }
gfCNCPoint3[27193] = {X 434.7568, Y 10.3819, Z -4.6667, A 0.000, B 0.000, C 0.000 }
gfCNCPoint3[27194] = {X 436.1450, Y 9.5742, Z -4.6667, A 0.000, B 0.000, C 0.000 }
gfCNCPoint3[27195] = {X 437.6322, Y 8.9676, Z -4.6667, A 0.000, B 0.000, C 0.000 }
gfCNCPoint3[27196] = {X 439.1893, Y 8.5739, Z -4.6667, A 0.000, B 0.000, C 0.000 }
gfCNCPoint3[27197] = {X 441.2579, Y 8.2873, Z -4.6667, A 0.000, B 0.000, C 0.000 }
gfCNCPoint3[27198] = {X 443.3442, Y 8.1946, Z -4.6667, A 0.000, B 0.000, C 0.000 }
gfCNCPoint3[27199] = {X 444.0367, Y 8.1906, Z -4.6667, A 0.000, B 0.000, C 0.000 }
gfCNCPoint3[27200] = {X 459.4467, Y 8.1906, Z -4.6667, A 0.000, B 0.000, C 0.000 }
gfCNCPoint3[27201] = {X 460.3348, Y 8.2906, Z -4.6667, A 0.000, B 0.000, C 0.000 }
gfCNCPoint3[27202] = {X 461.1784, Y 8.5858, Z -4.6667, A 0.000, B 0.000, C 0.000 }
gfCNCPoint3[27203] = {X 461.9352, Y 9.0613, Z -4.6667, A 0.000, B 0.000, C 0.000 }
gfCNCPoint3[27204] = {X 462.5672, Y 9.6933, Z -4.6667, A 0.000, B 0.000, C 0.000 }
gfCNCPoint3[27205] = {X 463.0427, Y 10.4501, Z -4.6667, A 0.000, B 0.000, C 0.000 }
gfCNCPoint3[27206] = {X 463.3379, Y 11.2937, Z -4.6667, A 0.000, B 0.000, C 0.000 }
gfCNCPoint3[27207] = {X 463.4379, Y 12.1818, Z -4.6667, A 0.000, B 0.000, C 0.000 }
gfCNCPoint3[27208] = {X 463.4378, Y 13.0163, Z -4.6667, A 0.000, B 0.000, C 0.000 }
gfCNCPoint3[27209] = {X 463.3397, Y 13.8589, Z -4.6667, A 0.000, B 0.000, C 0.000 }
gfCNCPoint3[27210] = {X 463.0662, Y 14.6619, Z -4.6667, A 0.000, B 0.000, C 0.000 }
gfCNCPoint3[27211] = {X 462.6296, Y 15.3891, Z -4.6667, A 0.000, B 0.000, C 0.000 }
gfCNCPoint3[27212] = {X 462.0494, Y 16.0080, Z -4.6667, A 0.000, B 0.000, C 0.000 }
gfCNCPoint3[27213] = {X 461.9726, Y 16.0725, Z -4.6667, A 0.000, B 0.000, C 0.000 }
gfCNCPoint3[27214] = {X 461.8942, Y 16.1351, Z -4.6667, A 0.000, B 0.000, C 0.000 }
gfCNCPoint3[27215] = {X 461.9106, Y 16.1930, Z -4.6667, A 0.000, B 0.000, C 0.000 }
gfCNCPoint3[27216] = {X 461.9100, Y 16.7687, Z -4.6667, A 0.000, B 0.000, C 0.000 }
gfCNCPoint3[27217] = {X 461.9105, Y 28.5935, Z -4.6667, A 0.000, B 0.000, C 0.000 }
gfCNCPoint3[27218] = {X 465.9908, Y 28.5933, Z -4.6667, A 0.000, B 0.000, C 0.000 }
gfCNCPoint3[27219] = {X 465.9908, Y 28.5933, Z -1.6667, A 0.000, B 0.000, C 0.000 }
gfCNCPoint3[27220] = {X 465.9908, Y 28.5933, Z 11.0000, A 0.000, B 0.000, C 0.000 }
gfCNCPoint3[27221] = {X 492.3835, Y 3.7906, Z 11.0000, A 0.000, B 0.000, C 0.000 }
gfCNCPoint3[27222] = {X 492.3835, Y 3.7906, Z -1.6667, A 0.000, B 0.000, C 0.000 }
gfCNCPoint3[27223] = {X 492.3835, Y 3.7906, Z -4.6667, A 0.000, B 0.000, C 0.000 }
gfCNCPoint3[27224] = {X 492.3835, Y 7.8706, Z -4.6667, A 0.000, B 0.000, C 0.000 }
gfCNCPoint3[27225] = {X 502.2066, Y 7.8706, Z -4.6667, A 0.000, B 0.000, C 0.000 }
gfCNCPoint3[27226] = {X 502.7394, Y 7.8747, Z -4.6667, A 0.000, B 0.000, C 0.000 }
gfCNCPoint3[27227] = {X 503.6913, Y 7.9890, Z -4.6667, A 0.000, B 0.000, C 0.000 }
gfCNCPoint3[27228] = {X 504.5943, Y 8.3112, Z -4.6667, A 0.000, B 0.000, C 0.000 }
gfCNCPoint3[27229] = {X 505.4035, Y 8.8253, Z -4.6667, A 0.000, B 0.000, C 0.000 }
gfCNCPoint3[27230] = {X 506.0787, Y 9.5059, Z -4.6667, A 0.000, B 0.000, C 0.000 }
gfCNCPoint3[27231] = {X 506.5865, Y 10.3191, Z -4.6667, A 0.000, B 0.000, C 0.000 }
gfCNCPoint3[27232] = {X 506.9017, Y 11.2245, Z -4.6667, A 0.000, B 0.000, C 0.000 }
gfCNCPoint3[27233] = {X 507.0085, Y 12.1773, Z -4.6667, A 0.000, B 0.000, C 0.000 }
gfCNCPoint3[27234] = {X 507.0085, Y 12.9782, Z -4.6667, A 0.000, B 0.000, C 0.000 }
gfCNCPoint3[27235] = {X 506.9072, Y 13.9081, Z -4.6667, A 0.000, B 0.000, C 0.000 }
gfCNCPoint3[27236] = {X 506.6081, Y 14.7944, Z -4.6667, A 0.000, B 0.000, C 0.000 }
gfCNCPoint3[27237] = {X 506.1252, Y 15.5955, Z -4.6667, A 0.000, B 0.000, C 0.000 }
gfCNCPoint3[27238] = {X 505.4812, Y 16.2740, Z -4.6667, A 0.000, B 0.000, C 0.000 }
gfCNCPoint3[27239] = {X 505.4811, Y 40.9128, Z -4.6667, A 0.000, B 0.000, C 0.000 }
gfCNCPoint3[27240] = {X 506.1195, Y 41.5838, Z -4.6667, A 0.000, B 0.000, C 0.000 }
gfCNCPoint3[27241] = {X 506.6002, Y 42.3755, Z -4.6667, A 0.000, B 0.000, C 0.000 }
gfCNCPoint3[27242] = {X 506.9011, Y 43.2514, Z -4.6667, A 0.000, B 0.000, C 0.000 }
gfCNCPoint3[27243] = {X 507.0083, Y 44.1713, Z -4.6667, A 0.000, B 0.000, C 0.000 }
gfCNCPoint3[27244] = {X 507.0085, Y 45.0000, Z -4.6667, A 0.000, B 0.000, C 0.000 }
gfCNCPoint3[27245] = {X 506.9002, Y 45.9613, Z -4.6667, A 0.000, B 0.000, C 0.000 }
gfCNCPoint3[27246] = {X 506.5807, Y 46.8744, Z -4.6667, A 0.000, B 0.000, C 0.000 }
gfCNCPoint3[27247] = {X 506.0660, Y 47.6935, Z -4.6667, A 0.000, B 0.000, C 0.000 }
gfCNCPoint3[27248] = {X 505.3820, Y 48.3775, Z -4.6667, A 0.000, B 0.000, C 0.000 }
gfCNCPoint3[27249] = {X 504.5629, Y 48.8922, Z -4.6667, A 0.000, B 0.000, C 0.000 }
gfCNCPoint3[27250] = {X 503.6498, Y 49.2117, Z -4.6667, A 0.000, B 0.000, C 0.000 }
gfCNCPoint3[27251] = {X 502.6885, Y 49.3200, Z -4.6667, A 0.000, B 0.000, C 0.000 }
gfCNCPoint3[27252] = {X 496.2450, Y 49.3200, Z -4.6667, A 0.000, B 0.000, C 0.000 }
gfCNCPoint3[27253] = {X 495.2885, Y 49.2128, Z -4.6667, A 0.000, B 0.000, C 0.000 }
gfCNCPoint3[27254] = {X 494.3794, Y 48.8964, Z -4.6667, A 0.000, B 0.000, C 0.000 }
gfCNCPoint3[27255] = {X 493.5630, Y 48.3866, Z -4.6667, A 0.000, B 0.000, C 0.000 }
gfCNCPoint3[27256] = {X 492.8797, Y 47.7087, Z -4.6667, A 0.000, B 0.000, C 0.000 }
gfCNCPoint3[27257] = {X 492.3635, Y 46.8963, Z -4.6667, A 0.000, B 0.000, C 0.000 }
gfCNCPoint3[27258] = {X 492.0399, Y 45.9898, Z -4.6667, A 0.000, B 0.000, C 0.000 }
gfCNCPoint3[27259] = {X 491.9252, Y 45.0341, Z -4.6667, A 0.000, B 0.000, C 0.000 }
gfCNCPoint3[27260] = {X 491.9254, Y 44.1494, Z -4.6667, A 0.000, B 0.000, C 0.000 }
gfCNCPoint3[27261] = {X 492.0359, Y 43.2364, Z -4.6667, A 0.000, B 0.000, C 0.000 }
gfCNCPoint3[27262] = {X 492.3371, Y 42.3675, Z -4.6667, A 0.000, B 0.000, C 0.000 }
gfCNCPoint3[27263] = {X 492.8153, Y 41.5821, Z -4.6667, A 0.000, B 0.000, C 0.000 }
gfCNCPoint3[27264] = {X 493.4490, Y 40.9157, Z -4.6667, A 0.000, B 0.000, C 0.000 }
gfCNCPoint3[27265] = {X 493.4490, Y 34.4738, Z -4.6667, A 0.000, B 0.000, C 0.000 }
gfCNCPoint3[27266] = {X 490.7245, Y 34.4738, Z -4.6667, A 0.000, B 0.000, C 0.000 }
gfCNCPoint3[27267] = {X 486.4401, Y 42.8168, Z -4.6667, A 0.000, B 0.000, C 0.000 }
gfCNCPoint3[27268] = {X 486.4450, Y 42.8299, Z -4.6667, A 0.000, B 0.000, C 0.000 }
gfCNCPoint3[27269] = {X 486.6110, Y 43.4909, Z -4.6667, A 0.000, B 0.000, C 0.000 }
gfCNCPoint3[27270] = {X 486.6708, Y 44.1699, Z -4.6667, A 0.000, B 0.000, C 0.000 }
gfCNCPoint3[27271] = {X 486.6710, Y 45.0000, Z -4.6667, A 0.000, B 0.000, C 0.000 }
gfCNCPoint3[27272] = {X 486.5627, Y 45.9613, Z -4.6667, A 0.000, B 0.000, C 0.000 }
gfCNCPoint3[27273] = {X 486.2432, Y 46.8744, Z -4.6667, A 0.000, B 0.000, C 0.000 }
gfCNCPoint3[27274] = {X 485.7285, Y 47.6935, Z -4.6667, A 0.000, B 0.000, C 0.000 }
gfCNCPoint3[27275] = {X 485.0445, Y 48.3775, Z -4.6667, A 0.000, B 0.000, C 0.000 }
gfCNCPoint3[27276] = {X 484.2254, Y 48.8922, Z -4.6667, A 0.000, B 0.000, C 0.000 }
gfCNCPoint3[27277] = {X 483.3123, Y 49.2117, Z -4.6667, A 0.000, B 0.000, C 0.000 }
gfCNCPoint3[27278] = {X 482.3510, Y 49.3200, Z -4.6667, A 0.000, B 0.000, C 0.000 }
gfCNCPoint3[27279] = {X 475.7650, Y 49.3200, Z -4.6667, A 0.000, B 0.000, C 0.000 }
gfCNCPoint3[27280] = {X 474.8037, Y 49.2117, Z -4.6667, A 0.000, B 0.000, C 0.000 }
gfCNCPoint3[27281] = {X 473.8906, Y 48.8922, Z -4.6667, A 0.000, B 0.000, C 0.000 }
gfCNCPoint3[27282] = {X 473.0715, Y 48.3775, Z -4.6667, A 0.000, B 0.000, C 0.000 }
gfCNCPoint3[27283] = {X 472.3875, Y 47.6935, Z -4.6667, A 0.000, B 0.000, C 0.000 }
gfCNCPoint3[27284] = {X 471.8728, Y 46.8744, Z -4.6667, A 0.000, B 0.000, C 0.000 }
gfCNCPoint3[27285] = {X 471.5533, Y 45.9614, Z -4.6667, A 0.000, B 0.000, C 0.000 }
gfCNCPoint3[27286] = {X 471.4450, Y 45.0001, Z -4.6667, A 0.000, B 0.000, C 0.000 }
gfCNCPoint3[27287] = {X 471.4454, Y 44.1494, Z -4.6667, A 0.000, B 0.000, C 0.000 }
gfCNCPoint3[27288] = {X 471.5430, Y 43.2935, Z -4.6667, A 0.000, B 0.000, C 0.000 }
gfCNCPoint3[27289] = {X 471.8086, Y 42.4740, Z -4.6667, A 0.000, B 0.000, C 0.000 }
gfCNCPoint3[27290] = {X 472.2314, Y 41.7236, Z -4.6667, A 0.000, B 0.000, C 0.000 }
gfCNCPoint3[27291] = {X 472.7947, Y 41.0719, Z -4.6667, A 0.000, B 0.000, C 0.000 }
gfCNCPoint3[27292] = {X 473.4762, Y 40.5449, Z -4.6667, A 0.000, B 0.000, C 0.000 }
gfCNCPoint3[27293] = {X 474.2486, Y 40.1637, Z -4.6667, A 0.000, B 0.000, C 0.000 }
gfCNCPoint3[27294] = {X 478.2331, Y 32.3645, Z -4.6667, A 0.000, B 0.000, C 0.000 }
gfCNCPoint3[27295] = {X 476.9696, Y 31.4969, Z -4.6667, A 0.000, B 0.000, C 0.000 }
gfCNCPoint3[27296] = {X 475.8331, Y 30.4685, Z -4.6667, A 0.000, B 0.000, C 0.000 }
gfCNCPoint3[27297] = {X 474.8439, Y 29.2978, Z -4.6667, A 0.000, B 0.000, C 0.000 }
gfCNCPoint3[27298] = {X 474.0196, Y 28.0057, Z -4.6667, A 0.000, B 0.000, C 0.000 }
gfCNCPoint3[27299] = {X 473.3750, Y 26.6152, Z -4.6667, A 0.000, B 0.000, C 0.000 }
gfCNCPoint3[27300] = {X 472.9215, Y 25.1511, Z -4.6667, A 0.000, B 0.000, C 0.000 }
gfCNCPoint3[27301] = {X 472.6072, Y 23.4680, Z -4.6667, A 0.000, B 0.000, C 0.000 }
gfCNCPoint3[27302] = {X 472.4666, Y 21.7616, Z -4.6667, A 0.000, B 0.000, C 0.000 }
gfCNCPoint3[27303] = {X 472.5013, Y 20.0498, Z -4.6667, A 0.000, B 0.000, C 0.000 }
gfCNCPoint3[27304] = {X 472.7109, Y 18.3505, Z -4.6667, A 0.000, B 0.000, C 0.000 }
gfCNCPoint3[27305] = {X 473.0932, Y 16.6815, Z -4.6667, A 0.000, B 0.000, C 0.000 }
gfCNCPoint3[27306] = {X 473.6359, Y 15.1666, Z -4.6667, A 0.000, B 0.000, C 0.000 }
gfCNCPoint3[27307] = {X 474.3792, Y 13.7394, Z -4.6667, A 0.000, B 0.000, C 0.000 }
gfCNCPoint3[27308] = {X 475.3093, Y 12.4263, Z -4.6667, A 0.000, B 0.000, C 0.000 }
gfCNCPoint3[27309] = {X 476.4090, Y 11.2515, Z -4.6667, A 0.000, B 0.000, C 0.000 }
gfCNCPoint3[27310] = {X 477.6579, Y 10.2368, Z -4.6667, A 0.000, B 0.000, C 0.000 }
gfCNCPoint3[27311] = {X 479.0330, Y 9.4010, Z -4.6667, A 0.000, B 0.000, C 0.000 }
gfCNCPoint3[27312] = {X 480.5087, Y 8.7595, Z -4.6667, A 0.000, B 0.000, C 0.000 }
gfCNCPoint3[27313] = {X 482.0579, Y 8.3242, Z -4.6667, A 0.000, B 0.000, C 0.000 }
gfCNCPoint3[27314] = {X 484.1552, Y 7.9974, Z -4.6667, A 0.000, B 0.000, C 0.000 }
gfCNCPoint3[27315] = {X 486.2748, Y 7.8827, Z -4.6667, A 0.000, B 0.000, C 0.000 }
gfCNCPoint3[27316] = {X 486.9679, Y 7.8706, Z -4.6667, A 0.000, B 0.000, C 0.000 }
gfCNCPoint3[27317] = {X 492.3835, Y 7.8706, Z -4.6667, A 0.000, B 0.000, C 0.000 }
gfCNCPoint3[27318] = {X 492.3835, Y 3.8706, Z -4.6667, A 0.000, B 0.000, C 0.000 }
gfCNCPoint3[27319] = {X 492.3835, Y 7.9506, Z -4.6667, A 0.000, B 0.000, C 0.000 }
gfCNCPoint3[27320] = {X 502.2063, Y 7.9506, Z -4.6667, A 0.000, B 0.000, C 0.000 }
gfCNCPoint3[27321] = {X 502.7388, Y 7.9547, Z -4.6667, A 0.000, B 0.000, C 0.000 }
gfCNCPoint3[27322] = {X 503.6730, Y 8.0669, Z -4.6667, A 0.000, B 0.000, C 0.000 }
gfCNCPoint3[27323] = {X 504.5592, Y 8.3831, Z -4.6667, A 0.000, B 0.000, C 0.000 }
gfCNCPoint3[27324] = {X 505.3533, Y 8.8876, Z -4.6667, A 0.000, B 0.000, C 0.000 }
gfCNCPoint3[27325] = {X 506.0160, Y 9.5555, Z -4.6667, A 0.000, B 0.000, C 0.000 }
gfCNCPoint3[27326] = {X 506.5144, Y 10.3536, Z -4.6667, A 0.000, B 0.000, C 0.000 }
gfCNCPoint3[27327] = {X 506.8237, Y 11.2422, Z -4.6667, A 0.000, B 0.000, C 0.000 }
gfCNCPoint3[27328] = {X 506.9285, Y 12.1773, Z -4.6667, A 0.000, B 0.000, C 0.000 }
gfCNCPoint3[27329] = {X 506.9285, Y 12.9782, Z -4.6667, A 0.000, B 0.000, C 0.000 }
gfCNCPoint3[27330] = {X 506.8271, Y 13.8999, Z -4.6667, A 0.000, B 0.000, C 0.000 }
gfCNCPoint3[27331] = {X 506.5277, Y 14.7775, Z -4.6667, A 0.000, B 0.000, C 0.000 }
gfCNCPoint3[27332] = {X 506.0447, Y 15.5690, Z -4.6667, A 0.000, B 0.000, C 0.000 }
gfCNCPoint3[27333] = {X 505.4012, Y 16.2367, Z -4.6667, A 0.000, B 0.000, C 0.000 }
gfCNCPoint3[27334] = {X 505.4011, Y 40.9506, Z -4.6667, A 0.000, B 0.000, C 0.000 }
gfCNCPoint3[27335] = {X 505.4294, Y 40.9738, Z -4.6667, A 0.000, B 0.000, C 0.000 }
gfCNCPoint3[27336] = {X 506.0560, Y 41.6324, Z -4.6667, A 0.000, B 0.000, C 0.000 }
gfCNCPoint3[27337] = {X 506.5277, Y 42.4094, Z -4.6667, A 0.000, B 0.000, C 0.000 }
gfCNCPoint3[27338] = {X 506.8231, Y 43.2691, Z -4.6667, A 0.000, B 0.000, C 0.000 }
gfCNCPoint3[27339] = {X 506.9283, Y 44.1720, Z -4.6667, A 0.000, B 0.000, C 0.000 }
gfCNCPoint3[27340] = {X 506.9285, Y 45.0000, Z -4.6667, A 0.000, B 0.000, C 0.000 }
gfCNCPoint3[27341] = {X 506.8222, Y 45.9435, Z -4.6667, A 0.000, B 0.000, C 0.000 }
gfCNCPoint3[27342] = {X 506.5086, Y 46.8397, Z -4.6667, A 0.000, B 0.000, C 0.000 }
gfCNCPoint3[27343] = {X 506.0035, Y 47.6436, Z -4.6667, A 0.000, B 0.000, C 0.000 }
gfCNCPoint3[27344] = {X 505.3321, Y 48.3150, Z -4.6667, A 0.000, B 0.000, C 0.000 }
gfCNCPoint3[27345] = {X 504.5282, Y 48.8201, Z -4.6667, A 0.000, B 0.000, C 0.000 }
gfCNCPoint3[27346] = {X 503.6320, Y 49.1337, Z -4.6667, A 0.000, B 0.000, C 0.000 }
gfCNCPoint3[27347] = {X 502.6885, Y 49.2400, Z -4.6667, A 0.000, B 0.000, C 0.000 }
gfCNCPoint3[27348] = {X 496.2450, Y 49.2400, Z -4.6667, A 0.000, B 0.000, C 0.000 }
gfCNCPoint3[27349] = {X 495.3062, Y 49.1348, Z -4.6667, A 0.000, B 0.000, C 0.000 }
gfCNCPoint3[27350] = {X 494.4140, Y 48.8242, Z -4.6667, A 0.000, B 0.000, C 0.000 }
gfCNCPoint3[27351] = {X 493.6127, Y 48.3239, Z -4.6667, A 0.000, B 0.000, C 0.000 }
gfCNCPoint3[27352] = {X 492.9420, Y 47.6585, Z -4.6667, A 0.000, B 0.000, C 0.000 }
gfCNCPoint3[27353] = {X 492.4354, Y 46.8612, Z -4.6667, A 0.000, B 0.000, C 0.000 }
gfCNCPoint3[27354] = {X 492.1178, Y 45.9714, Z -4.6667, A 0.000, B 0.000, C 0.000 }
gfCNCPoint3[27355] = {X 492.0052, Y 45.0335, Z -4.6667, A 0.000, B 0.000, C 0.000 }
gfCNCPoint3[27356] = {X 492.0054, Y 44.1505, Z -4.6667, A 0.000, B 0.000, C 0.000 }
gfCNCPoint3[27357] = {X 492.1159, Y 43.2454, Z -4.6667, A 0.000, B 0.000, C 0.000 }
gfCNCPoint3[27358] = {X 492.4173, Y 42.3850, Z -4.6667, A 0.000, B 0.000, C 0.000 }
gfCNCPoint3[27359] = {X 492.8957, Y 41.6088, Z -4.6667, A 0.000, B 0.000, C 0.000 }
gfCNCPoint3[27360] = {X 493.5290, Y 40.9529, Z -4.6667, A 0.000, B 0.000, C 0.000 }
gfCNCPoint3[27361] = {X 493.5290, Y 34.3938, Z -4.6667, A 0.000, B 0.000, C 0.000 }
gfCNCPoint3[27362] = {X 490.6756, Y 34.3938, Z -4.6667, A 0.000, B 0.000, C 0.000 }
gfCNCPoint3[27363] = {X 486.3528, Y 42.8118, Z -4.6667, A 0.000, B 0.000, C 0.000 }
gfCNCPoint3[27364] = {X 486.3697, Y 42.8567, Z -4.6667, A 0.000, B 0.000, C 0.000 }
gfCNCPoint3[27365] = {X 486.5322, Y 43.5049, Z -4.6667, A 0.000, B 0.000, C 0.000 }
gfCNCPoint3[27366] = {X 486.5908, Y 44.1706, Z -4.6667, A 0.000, B 0.000, C 0.000 }
gfCNCPoint3[27367] = {X 486.5910, Y 45.0000, Z -4.6667, A 0.000, B 0.000, C 0.000 }
gfCNCPoint3[27368] = {X 486.4847, Y 45.9435, Z -4.6667, A 0.000, B 0.000, C 0.000 }
gfCNCPoint3[27369] = {X 486.1711, Y 46.8397, Z -4.6667, A 0.000, B 0.000, C 0.000 }
gfCNCPoint3[27370] = {X 485.6660, Y 47.6436, Z -4.6667, A 0.000, B 0.000, C 0.000 }
gfCNCPoint3[27371] = {X 484.9946, Y 48.3150, Z -4.6667, A 0.000, B 0.000, C 0.000 }
gfCNCPoint3[27372] = {X 484.1907, Y 48.8201, Z -4.6667, A 0.000, B 0.000, C 0.000 }
gfCNCPoint3[27373] = {X 483.2945, Y 49.1337, Z -4.6667, A 0.000, B 0.000, C 0.000 }
gfCNCPoint3[27374] = {X 482.3510, Y 49.2400, Z -4.6667, A 0.000, B 0.000, C 0.000 }
gfCNCPoint3[27375] = {X 475.7650, Y 49.2400, Z -4.6667, A 0.000, B 0.000, C 0.000 }
gfCNCPoint3[27376] = {X 474.8215, Y 49.1337, Z -4.6667, A 0.000, B 0.000, C 0.000 }
gfCNCPoint3[27377] = {X 473.9253, Y 48.8201, Z -4.6667, A 0.000, B 0.000, C 0.000 }
gfCNCPoint3[27378] = {X 473.1214, Y 48.3150, Z -4.6667, A 0.000, B 0.000, C 0.000 }
gfCNCPoint3[27379] = {X 472.4500, Y 47.6436, Z -4.6667, A 0.000, B 0.000, C 0.000 }
gfCNCPoint3[27380] = {X 471.9449, Y 46.8397, Z -4.6667, A 0.000, B 0.000, C 0.000 }
gfCNCPoint3[27381] = {X 471.6313, Y 45.9436, Z -4.6667, A 0.000, B 0.000, C 0.000 }
gfCNCPoint3[27382] = {X 471.5250, Y 45.0001, Z -4.6667, A 0.000, B 0.000, C 0.000 }
gfCNCPoint3[27383] = {X 471.5254, Y 44.1505, Z -4.6667, A 0.000, B 0.000, C 0.000 }
gfCNCPoint3[27384] = {X 471.6223, Y 43.3054, Z -4.6667, A 0.000, B 0.000, C 0.000 }
gfCNCPoint3[27385] = {X 471.8860, Y 42.4967, Z -4.6667, A 0.000, B 0.000, C 0.000 }
gfCNCPoint3[27386] = {X 472.3057, Y 41.7570, Z -4.6667, A 0.000, B 0.000, C 0.000 }
gfCNCPoint3[27387] = {X 472.8647, Y 41.1158, Z -4.6667, A 0.000, B 0.000, C 0.000 }
gfCNCPoint3[27388] = {X 473.5404, Y 40.5992, Z -4.6667, A 0.000, B 0.000, C 0.000 }
gfCNCPoint3[27389] = {X 474.3057, Y 40.2278, Z -4.6667, A 0.000, B 0.000, C 0.000 }
gfCNCPoint3[27390] = {X 478.3386, Y 32.3338, Z -4.6667, A 0.000, B 0.000, C 0.000 }
gfCNCPoint3[27391] = {X 477.0684, Y 31.4728, Z -4.6667, A 0.000, B 0.000, C 0.000 }
gfCNCPoint3[27392] = {X 475.9255, Y 30.4488, Z -4.6667, A 0.000, B 0.000, C 0.000 }
gfCNCPoint3[27393] = {X 474.9306, Y 29.2805, Z -4.6667, A 0.000, B 0.000, C 0.000 }
gfCNCPoint3[27394] = {X 474.1018, Y 27.9891, Z -4.6667, A 0.000, B 0.000, C 0.000 }
gfCNCPoint3[27395] = {X 473.4541, Y 26.5980, Z -4.6667, A 0.000, B 0.000, C 0.000 }
gfCNCPoint3[27396] = {X 472.9992, Y 25.1324, Z -4.6667, A 0.000, B 0.000, C 0.000 }
gfCNCPoint3[27397] = {X 472.6865, Y 23.4574, Z -4.6667, A 0.000, B 0.000, C 0.000 }
gfCNCPoint3[27398] = {X 472.5466, Y 21.7591, Z -4.6667, A 0.000, B 0.000, C 0.000 }
gfCNCPoint3[27399] = {X 472.5811, Y 20.0555, Z -4.6667, A 0.000, B 0.000, C 0.000 }
gfCNCPoint3[27400] = {X 472.7897, Y 18.3643, Z -4.6667, A 0.000, B 0.000, C 0.000 }
gfCNCPoint3[27401] = {X 473.1701, Y 16.7033, Z -4.6667, A 0.000, B 0.000, C 0.000 }
gfCNCPoint3[27402] = {X 473.7092, Y 15.1987, Z -4.6667, A 0.000, B 0.000, C 0.000 }
gfCNCPoint3[27403] = {X 474.4475, Y 13.7811, Z -4.6667, A 0.000, B 0.000, C 0.000 }
gfCNCPoint3[27404] = {X 475.3713, Y 12.4769, Z -4.6667, A 0.000, B 0.000, C 0.000 }
gfCNCPoint3[27405] = {X 476.4635, Y 11.3100, Z -4.6667, A 0.000, B 0.000, C 0.000 }
gfCNCPoint3[27406] = {X 477.7040, Y 10.3022, Z -4.6667, A 0.000, B 0.000, C 0.000 }
gfCNCPoint3[27407] = {X 479.0698, Y 9.4721, Z -4.6667, A 0.000, B 0.000, C 0.000 }
gfCNCPoint3[27408] = {X 480.5355, Y 8.8349, Z -4.6667, A 0.000, B 0.000, C 0.000 }
gfCNCPoint3[27409] = {X 482.0742, Y 8.4025, Z -4.6667, A 0.000, B 0.000, C 0.000 }
gfCNCPoint3[27410] = {X 484.1638, Y 8.0769, Z -4.6667, A 0.000, B 0.000, C 0.000 }
gfCNCPoint3[27411] = {X 486.2756, Y 7.9627, Z -4.6667, A 0.000, B 0.000, C 0.000 }
gfCNCPoint3[27412] = {X 486.9686, Y 7.9506, Z -4.6667, A 0.000, B 0.000, C 0.000 }
gfCNCPoint3[27413] = {X 492.3835, Y 7.9506, Z -4.6667, A 0.000, B 0.000, C 0.000 }
gfCNCPoint3[27414] = {X 492.3835, Y 3.9506, Z -4.6667, A 0.000, B 0.000, C 0.000 }
gfCNCPoint3[27415] = {X 492.3835, Y 8.0306, Z -4.6667, A 0.000, B 0.000, C 0.000 }
gfCNCPoint3[27416] = {X 502.2059, Y 8.0306, Z -4.6667, A 0.000, B 0.000, C 0.000 }
gfCNCPoint3[27417] = {X 502.7382, Y 8.0347, Z -4.6667, A 0.000, B 0.000, C 0.000 }
gfCNCPoint3[27418] = {X 503.6547, Y 8.1447, Z -4.6667, A 0.000, B 0.000, C 0.000 }
gfCNCPoint3[27419] = {X 504.5241, Y 8.4549, Z -4.6667, A 0.000, B 0.000, C 0.000 }
gfCNCPoint3[27420] = {X 505.3032, Y 8.9500, Z -4.6667, A 0.000, B 0.000, C 0.000 }
gfCNCPoint3[27421] = {X 505.9533, Y 9.6052, Z -4.6667, A 0.000, B 0.000, C 0.000 }
gfCNCPoint3[27422] = {X 506.4422, Y 10.3882, Z -4.6667, A 0.000, B 0.000, C 0.000 }
gfCNCPoint3[27423] = {X 506.7457, Y 11.2599, Z -4.6667, A 0.000, B 0.000, C 0.000 }
gfCNCPoint3[27424] = {X 506.8485, Y 12.1773, Z -4.6667, A 0.000, B 0.000, C 0.000 }
gfCNCPoint3[27425] = {X 506.8485, Y 12.9782, Z -4.6667, A 0.000, B 0.000, C 0.000 }
gfCNCPoint3[27426] = {X 506.7469, Y 13.8916, Z -4.6667, A 0.000, B 0.000, C 0.000 }
gfCNCPoint3[27427] = {X 506.4473, Y 14.7604, Z -4.6667, A 0.000, B 0.000, C 0.000 }
gfCNCPoint3[27428] = {X 505.9642, Y 15.5423, Z -4.6667, A 0.000, B 0.000, C 0.000 }
gfCNCPoint3[27429] = {X 505.3212, Y 16.1990, Z -4.6667, A 0.000, B 0.000, C 0.000 }
gfCNCPoint3[27430] = {X 505.3211, Y 40.9889, Z -4.6667, A 0.000, B 0.000, C 0.000 }
gfCNCPoint3[27431] = {X 505.3679, Y 41.0266, Z -4.6667, A 0.000, B 0.000, C 0.000 }
gfCNCPoint3[27432] = {X 505.9866, Y 41.6734, Z -4.6667, A 0.000, B 0.000, C 0.000 }
gfCNCPoint3[27433] = {X 506.4526, Y 42.4375, Z -4.6667, A 0.000, B 0.000, C 0.000 }
gfCNCPoint3[27434] = {X 506.7443, Y 43.2837, Z -4.6667, A 0.000, B 0.000, C 0.000 }
gfCNCPoint3[27435] = {X 506.8483, Y 44.1727, Z -4.6667, A 0.000, B 0.000, C 0.000 }
gfCNCPoint3[27436] = {X 506.8485, Y 45.0000, Z -4.6667, A 0.000, B 0.000, C 0.000 }
gfCNCPoint3[27437] = {X 506.7442, Y 45.9257, Z -4.6667, A 0.000, B 0.000, C 0.000 }
gfCNCPoint3[27438] = {X 506.4365, Y 46.8050, Z -4.6667, A 0.000, B 0.000, C 0.000 }
gfCNCPoint3[27439] = {X 505.9409, Y 47.5937, Z -4.6667, A 0.000, B 0.000, C 0.000 }
gfCNCPoint3[27440] = {X 505.2822, Y 48.2524, Z -4.6667, A 0.000, B 0.000, C 0.000 }
gfCNCPoint3[27441] = {X 504.4934, Y 48.7480, Z -4.6667, A 0.000, B 0.000, C 0.000 }
gfCNCPoint3[27442] = {X 503.6142, Y 49.0557, Z -4.6667, A 0.000, B 0.000, C 0.000 }
gfCNCPoint3[27443] = {X 502.6885, Y 49.1600, Z -4.6667, A 0.000, B 0.000, C 0.000 }
gfCNCPoint3[27444] = {X 496.2450, Y 49.1600, Z -4.6667, A 0.000, B 0.000, C 0.000 }
gfCNCPoint3[27445] = {X 495.3239, Y 49.0567, Z -4.6667, A 0.000, B 0.000, C 0.000 }
gfCNCPoint3[27446] = {X 494.4485, Y 48.7521, Z -4.6667, A 0.000, B 0.000, C 0.000 }
gfCNCPoint3[27447] = {X 493.6623, Y 48.2612, Z -4.6667, A 0.000, B 0.000, C 0.000 }
gfCNCPoint3[27448] = {X 493.0043, Y 47.6084, Z -4.6667, A 0.000, B 0.000, C 0.000 }
gfCNCPoint3[27449] = {X 492.5072, Y 46.8261, Z -4.6667, A 0.000, B 0.000, C 0.000 }
gfCNCPoint3[27450] = {X 492.1957, Y 45.9531, Z -4.6667, A 0.000, B 0.000, C 0.000 }
gfCNCPoint3[27451] = {X 492.0852, Y 45.0328, Z -4.6667, A 0.000, B 0.000, C 0.000 }
gfCNCPoint3[27452] = {X 492.0854, Y 44.1516, Z -4.6667, A 0.000, B 0.000, C 0.000 }
gfCNCPoint3[27453] = {X 492.1960, Y 43.2545, Z -4.6667, A 0.000, B 0.000, C 0.000 }
gfCNCPoint3[27454] = {X 492.4976, Y 42.4026, Z -4.6667, A 0.000, B 0.000, C 0.000 }
gfCNCPoint3[27455] = {X 492.9762, Y 41.6358, Z -4.6667, A 0.000, B 0.000, C 0.000 }
gfCNCPoint3[27456] = {X 493.6090, Y 40.9906, Z -4.6667, A 0.000, B 0.000, C 0.000 }
gfCNCPoint3[27457] = {X 493.6090, Y 34.3138, Z -4.6667, A 0.000, B 0.000, C 0.000 }
gfCNCPoint3[27458] = {X 490.6268, Y 34.3138, Z -4.6667, A 0.000, B 0.000, C 0.000 }
gfCNCPoint3[27459] = {X 486.2655, Y 42.8067, Z -4.6667, A 0.000, B 0.000, C 0.000 }
gfCNCPoint3[27460] = {X 486.2943, Y 42.8835, Z -4.6667, A 0.000, B 0.000, C 0.000 }
gfCNCPoint3[27461] = {X 486.4534, Y 43.5188, Z -4.6667, A 0.000, B 0.000, C 0.000 }
gfCNCPoint3[27462] = {X 486.5109, Y 44.1713, Z -4.6667, A 0.000, B 0.000, C 0.000 }
gfCNCPoint3[27463] = {X 486.5110, Y 45.0000, Z -4.6667, A 0.000, B 0.000, C 0.000 }
gfCNCPoint3[27464] = {X 486.4067, Y 45.9257, Z -4.6667, A 0.000, B 0.000, C 0.000 }
gfCNCPoint3[27465] = {X 486.0990, Y 46.8050, Z -4.6667, A 0.000, B 0.000, C 0.000 }
gfCNCPoint3[27466] = {X 485.6034, Y 47.5937, Z -4.6667, A 0.000, B 0.000, C 0.000 }
gfCNCPoint3[27467] = {X 484.9447, Y 48.2524, Z -4.6667, A 0.000, B 0.000, C 0.000 }
gfCNCPoint3[27468] = {X 484.1560, Y 48.7480, Z -4.6667, A 0.000, B 0.000, C 0.000 }
gfCNCPoint3[27469] = {X 483.2767, Y 49.0557, Z -4.6667, A 0.000, B 0.000, C 0.000 }
gfCNCPoint3[27470] = {X 482.3510, Y 49.1600, Z -4.6667, A 0.000, B 0.000, C 0.000 }
gfCNCPoint3[27471] = {X 475.7650, Y 49.1600, Z -4.6667, A 0.000, B 0.000, C 0.000 }
gfCNCPoint3[27472] = {X 474.8393, Y 49.0557, Z -4.6667, A 0.000, B 0.000, C 0.000 }
gfCNCPoint3[27473] = {X 473.9600, Y 48.7480, Z -4.6667, A 0.000, B 0.000, C 0.000 }
gfCNCPoint3[27474] = {X 473.1713, Y 48.2524, Z -4.6667, A 0.000, B 0.000, C 0.000 }
gfCNCPoint3[27475] = {X 472.5126, Y 47.5937, Z -4.6667, A 0.000, B 0.000, C 0.000 }
gfCNCPoint3[27476] = {X 472.0169, Y 46.8050, Z -4.6667, A 0.000, B 0.000, C 0.000 }
gfCNCPoint3[27477] = {X 471.7093, Y 45.9257, Z -4.6667, A 0.000, B 0.000, C 0.000 }
gfCNCPoint3[27478] = {X 471.6050, Y 45.0000, Z -4.6667, A 0.000, B 0.000, C 0.000 }
gfCNCPoint3[27479] = {X 471.6054, Y 44.1516, Z -4.6667, A 0.000, B 0.000, C 0.000 }
gfCNCPoint3[27480] = {X 471.7016, Y 43.3174, Z -4.6667, A 0.000, B 0.000, C 0.000 }
gfCNCPoint3[27481] = {X 471.9634, Y 42.5195, Z -4.6667, A 0.000, B 0.000, C 0.000 }
gfCNCPoint3[27482] = {X 472.3801, Y 41.7905, Z -4.6667, A 0.000, B 0.000, C 0.000 }
gfCNCPoint3[27483] = {X 472.9347, Y 41.1600, Z -4.6667, A 0.000, B 0.000, C 0.000 }
gfCNCPoint3[27484] = {X 473.6046, Y 40.6537, Z -4.6667, A 0.000, B 0.000, C 0.000 }
gfCNCPoint3[27485] = {X 474.3626, Y 40.2923, Z -4.6667, A 0.000, B 0.000, C 0.000 }
gfCNCPoint3[27486] = {X 478.4444, Y 32.3026, Z -4.6667, A 0.000, B 0.000, C 0.000 }
gfCNCPoint3[27487] = {X 477.1674, Y 31.4484, Z -4.6667, A 0.000, B 0.000, C 0.000 }
gfCNCPoint3[27488] = {X 476.0180, Y 30.4290, Z -4.6667, A 0.000, B 0.000, C 0.000 }
gfCNCPoint3[27489] = {X 475.0174, Y 29.2632, Z -4.6667, A 0.000, B 0.000, C 0.000 }
gfCNCPoint3[27490] = {X 474.1840, Y 27.9725, Z -4.6667, A 0.000, B 0.000, C 0.000 }
gfCNCPoint3[27491] = {X 473.5332, Y 26.5809, Z -4.6667, A 0.000, B 0.000, C 0.000 }
gfCNCPoint3[27492] = {X 473.0770, Y 25.1138, Z -4.6667, A 0.000, B 0.000, C 0.000 }
gfCNCPoint3[27493] = {X 472.7658, Y 23.4468, Z -4.6667, A 0.000, B 0.000, C 0.000 }
gfCNCPoint3[27494] = {X 472.6266, Y 21.7567, Z -4.6667, A 0.000, B 0.000, C 0.000 }
gfCNCPoint3[27495] = {X 472.6609, Y 20.0612, Z -4.6667, A 0.000, B 0.000, C 0.000 }
gfCNCPoint3[27496] = {X 472.8685, Y 18.3781, Z -4.6667, A 0.000, B 0.000, C 0.000 }
gfCNCPoint3[27497] = {X 473.2471, Y 16.7251, Z -4.6667, A 0.000, B 0.000, C 0.000 }
gfCNCPoint3[27498] = {X 473.7825, Y 15.2307, Z -4.6667, A 0.000, B 0.000, C 0.000 }
gfCNCPoint3[27499] = {X 474.5158, Y 13.8228, Z -4.6667, A 0.000, B 0.000, C 0.000 }
gfCNCPoint3[27500] = {X 475.4333, Y 12.5274, Z -4.6667, A 0.000, B 0.000, C 0.000 }
gfCNCPoint3[27501] = {X 476.5181, Y 11.3686, Z -4.6667, A 0.000, B 0.000, C 0.000 }
gfCNCPoint3[27502] = {X 477.7501, Y 10.3676, Z -4.6667, A 0.000, B 0.000, C 0.000 }
gfCNCPoint3[27503] = {X 479.1066, Y 9.5431, Z -4.6667, A 0.000, B 0.000, C 0.000 }
gfCNCPoint3[27504] = {X 480.5624, Y 8.9103, Z -4.6667, A 0.000, B 0.000, C 0.000 }
gfCNCPoint3[27505] = {X 482.0906, Y 8.4808, Z -4.6667, A 0.000, B 0.000, C 0.000 }
gfCNCPoint3[27506] = {X 484.1725, Y 8.1564, Z -4.6667, A 0.000, B 0.000, C 0.000 }
gfCNCPoint3[27507] = {X 486.2765, Y 8.0427, Z -4.6667, A 0.000, B 0.000, C 0.000 }
gfCNCPoint3[27508] = {X 486.9693, Y 8.0306, Z -4.6667, A 0.000, B 0.000, C 0.000 }
gfCNCPoint3[27509] = {X 492.3835, Y 8.0306, Z -4.6667, A 0.000, B 0.000, C 0.000 }
gfCNCPoint3[27510] = {X 492.3835, Y 4.0306, Z -4.6667, A 0.000, B 0.000, C 0.000 }
gfCNCPoint3[27511] = {X 492.3835, Y 8.1106, Z -4.6667, A 0.000, B 0.000, C 0.000 }
gfCNCPoint3[27512] = {X 502.2056, Y 8.1106, Z -4.6667, A 0.000, B 0.000, C 0.000 }
gfCNCPoint3[27513] = {X 502.7376, Y 8.1147, Z -4.6667, A 0.000, B 0.000, C 0.000 }
gfCNCPoint3[27514] = {X 503.6364, Y 8.2226, Z -4.6667, A 0.000, B 0.000, C 0.000 }
gfCNCPoint3[27515] = {X 504.4889, Y 8.5268, Z -4.6667, A 0.000, B 0.000, C 0.000 }
gfCNCPoint3[27516] = {X 505.2530, Y 9.0123, Z -4.6667, A 0.000, B 0.000, C 0.000 }
gfCNCPoint3[27517] = {X 505.8906, Y 9.6549, Z -4.6667, A 0.000, B 0.000, C 0.000 }
gfCNCPoint3[27518] = {X 506.3701, Y 10.4227, Z -4.6667, A 0.000, B 0.000, C 0.000 }
gfCNCPoint3[27519] = {X 506.6676, Y 11.2777, Z -4.6667, A 0.000, B 0.000, C 0.000 }
gfCNCPoint3[27520] = {X 506.7685, Y 12.1773, Z -4.6667, A 0.000, B 0.000, C 0.000 }
gfCNCPoint3[27521] = {X 506.7685, Y 12.9782, Z -4.6667, A 0.000, B 0.000, C 0.000 }
gfCNCPoint3[27522] = {X 506.6668, Y 13.8832, Z -4.6667, A 0.000, B 0.000, C 0.000 }
gfCNCPoint3[27523] = {X 506.3669, Y 14.7432, Z -4.6667, A 0.000, B 0.000, C 0.000 }
gfCNCPoint3[27524] = {X 505.8836, Y 15.5152, Z -4.6667, A 0.000, B 0.000, C 0.000 }
gfCNCPoint3[27525] = {X 505.2412, Y 16.1608, Z -4.6667, A 0.000, B 0.000, C 0.000 }
gfCNCPoint3[27526] = {X 505.2411, Y 41.0272, Z -4.6667, A 0.000, B 0.000, C 0.000 }
gfCNCPoint3[27527] = {X 505.3177, Y 41.0889, Z -4.6667, A 0.000, B 0.000, C 0.000 }
gfCNCPoint3[27528] = {X 505.9239, Y 41.7232, Z -4.6667, A 0.000, B 0.000, C 0.000 }
gfCNCPoint3[27529] = {X 506.3805, Y 42.4724, Z -4.6667, A 0.000, B 0.000, C 0.000 }
gfCNCPoint3[27530] = {X 506.6664, Y 43.3019, Z -4.6667, A 0.000, B 0.000, C 0.000 }
gfCNCPoint3[27531] = {X 506.7683, Y 44.1734, Z -4.6667, A 0.000, B 0.000, C 0.000 }
gfCNCPoint3[27532] = {X 506.7685, Y 45.0000, Z -4.6667, A 0.000, B 0.000, C 0.000 }
gfCNCPoint3[27533] = {X 506.6662, Y 45.9079, Z -4.6667, A 0.000, B 0.000, C 0.000 }
gfCNCPoint3[27534] = {X 506.3644, Y 46.7702, Z -4.6667, A 0.000, B 0.000, C 0.000 }
gfCNCPoint3[27535] = {X 505.8784, Y 47.5438, Z -4.6667, A 0.000, B 0.000, C 0.000 }
gfCNCPoint3[27536] = {X 505.2323, Y 48.1899, Z -4.6667, A 0.000, B 0.000, C 0.000 }
gfCNCPoint3[27537] = {X 504.4587, Y 48.6760, Z -4.6667, A 0.000, B 0.000, C 0.000 }
gfCNCPoint3[27538] = {X 503.5964, Y 48.9777, Z -4.6667, A 0.000, B 0.000, C 0.000 }
gfCNCPoint3[27539] = {X 502.6885, Y 49.0800, Z -4.6667, A 0.000, B 0.000, C 0.000 }
gfCNCPoint3[27540] = {X 496.2450, Y 49.0800, Z -4.6667, A 0.000, B 0.000, C 0.000 }
gfCNCPoint3[27541] = {X 495.3416, Y 48.9787, Z -4.6667, A 0.000, B 0.000, C 0.000 }
gfCNCPoint3[27542] = {X 494.4831, Y 48.6799, Z -4.6667, A 0.000, B 0.000, C 0.000 }
gfCNCPoint3[27543] = {X 493.7120, Y 48.1985, Z -4.6667, A 0.000, B 0.000, C 0.000 }
gfCNCPoint3[27544] = {X 493.0667, Y 47.5582, Z -4.6667, A 0.000, B 0.000, C 0.000 }
gfCNCPoint3[27545] = {X 492.5791, Y 46.7909, Z -4.6667, A 0.000, B 0.000, C 0.000 }
gfCNCPoint3[27546] = {X 492.2736, Y 45.9348, Z -4.6667, A 0.000, B 0.000, C 0.000 }
gfCNCPoint3[27547] = {X 492.1652, Y 45.0322, Z -4.6667, A 0.000, B 0.000, C 0.000 }
gfCNCPoint3[27548] = {X 492.1654, Y 44.1527, Z -4.6667, A 0.000, B 0.000, C 0.000 }
gfCNCPoint3[27549] = {X 492.2760, Y 43.2637, Z -4.6667, A 0.000, B 0.000, C 0.000 }
gfCNCPoint3[27550] = {X 492.5779, Y 42.4203, Z -4.6667, A 0.000, B 0.000, C 0.000 }
gfCNCPoint3[27551] = {X 493.0566, Y 41.6631, Z -4.6667, A 0.000, B 0.000, C 0.000 }
gfCNCPoint3[27552] = {X 493.6890, Y 41.0287, Z -4.6667, A 0.000, B 0.000, C 0.000 }
gfCNCPoint3[27553] = {X 493.6890, Y 34.2338, Z -4.6667, A 0.000, B 0.000, C 0.000 }
gfCNCPoint3[27554] = {X 490.5779, Y 34.2338, Z -4.6667, A 0.000, B 0.000, C 0.000 }
gfCNCPoint3[27555] = {X 486.1781, Y 42.8016, Z -4.6667, A 0.000, B 0.000, C 0.000 }
gfCNCPoint3[27556] = {X 486.2189, Y 42.9103, Z -4.6667, A 0.000, B 0.000, C 0.000 }
gfCNCPoint3[27557] = {X 486.3746, Y 43.5328, Z -4.6667, A 0.000, B 0.000, C 0.000 }
gfCNCPoint3[27558] = {X 486.4309, Y 44.1720, Z -4.6667, A 0.000, B 0.000, C 0.000 }
gfCNCPoint3[27559] = {X 486.4310, Y 45.0000, Z -4.6667, A 0.000, B 0.000, C 0.000 }
gfCNCPoint3[27560] = {X 486.3287, Y 45.9079, Z -4.6667, A 0.000, B 0.000, C 0.000 }
gfCNCPoint3[27561] = {X 486.0270, Y 46.7702, Z -4.6667, A 0.000, B 0.000, C 0.000 }
gfCNCPoint3[27562] = {X 485.5409, Y 47.5438, Z -4.6667, A 0.000, B 0.000, C 0.000 }
gfCNCPoint3[27563] = {X 484.8949, Y 48.1899, Z -4.6667, A 0.000, B 0.000, C 0.000 }
gfCNCPoint3[27564] = {X 484.1213, Y 48.6760, Z -4.6667, A 0.000, B 0.000, C 0.000 }
gfCNCPoint3[27565] = {X 483.2589, Y 48.9777, Z -4.6667, A 0.000, B 0.000, C 0.000 }
gfCNCPoint3[27566] = {X 482.3510, Y 49.0800, Z -4.6667, A 0.000, B 0.000, C 0.000 }
gfCNCPoint3[27567] = {X 475.7650, Y 49.0800, Z -4.6667, A 0.000, B 0.000, C 0.000 }
gfCNCPoint3[27568] = {X 474.8571, Y 48.9777, Z -4.6667, A 0.000, B 0.000, C 0.000 }
gfCNCPoint3[27569] = {X 473.9947, Y 48.6760, Z -4.6667, A 0.000, B 0.000, C 0.000 }
gfCNCPoint3[27570] = {X 473.2211, Y 48.1899, Z -4.6667, A 0.000, B 0.000, C 0.000 }
gfCNCPoint3[27571] = {X 472.5751, Y 47.5438, Z -4.6667, A 0.000, B 0.000, C 0.000 }
gfCNCPoint3[27572] = {X 472.0890, Y 46.7702, Z -4.6667, A 0.000, B 0.000, C 0.000 }
gfCNCPoint3[27573] = {X 471.7873, Y 45.9079, Z -4.6667, A 0.000, B 0.000, C 0.000 }
gfCNCPoint3[27574] = {X 471.6850, Y 45.0000, Z -4.6667, A 0.000, B 0.000, C 0.000 }
gfCNCPoint3[27575] = {X 471.6853, Y 44.1527, Z -4.6667, A 0.000, B 0.000, C 0.000 }
gfCNCPoint3[27576] = {X 471.7809, Y 43.3294, Z -4.6667, A 0.000, B 0.000, C 0.000 }
gfCNCPoint3[27577] = {X 472.0408, Y 42.5424, Z -4.6667, A 0.000, B 0.000, C 0.000 }
gfCNCPoint3[27578] = {X 472.4544, Y 41.8242, Z -4.6667, A 0.000, B 0.000, C 0.000 }
gfCNCPoint3[27579] = {X 473.0046, Y 41.2044, Z -4.6667, A 0.000, B 0.000, C 0.000 }
gfCNCPoint3[27580] = {X 473.6687, Y 40.7085, Z -4.6667, A 0.000, B 0.000, C 0.000 }
